// TIA Portal project "FischerTechnik_Origional_program_V16_V17" (V17)

(* hardware
DEVICE "ET 200SP-Station_1"  ET 200SP-Station
   slot 0: "Baugruppenträger_0"  Rack  6ES5 710-8MAx1
   slot 1: "PLC"  CPU 1512SP F-1 PN  6ES7 512-1SK01-0AB0  V2.8
      slot 32768: "PROFINET"  X1
         slot 32771: "Port_3"  X1 P3
   slot 2: "DO1+2"  DQ 16x24VDC/0.5A ST  6ES7 132-6BH01-0BA0  V0.0
      slot 1: "DO1+2"  DQ 16x24VDC/0.5A ST
   slot 3: "DO3+4"  DQ 16x24VDC/0.5A ST  6ES7 132-6BH01-0BA0  V0.0
      slot 1: "DO3+4"  DQ 16x24VDC/0.5A ST
   slot 4: "DO5"  DQ 8x24VDC/0.5A HF  6ES7 132-6BF00-0CA0  V2.0
      slot 1: "DO5"  DQ 8x24VDC/0.5A HF
   slot 5: "DO6"  DQ 8x24VDC/0.5A HF  6ES7 132-6BF00-0CA0  V2.0
      slot 1: "DO6"  DQ 8x24VDC/0.5A HF
   slot 6: "DO7-14"  DQ 4x24VDC/2A HS  6ES7 132-6BD20-0DA0  V2.0
      slot 1: "DO7-14"  DQ 4x24VDC/2A HS
   slot 7: "DO15-22"  DQ 4x24VDC/2A HS  6ES7 132-6BD20-0DA0  V2.0
      slot 1: "DO15-22"  DQ 4x24VDC/2A HS
   slot 8: "DO23-30"  DQ 4x24VDC/2A HS  6ES7 132-6BD20-0DA0  V2.0
      slot 1: "DO23-30"  DQ 4x24VDC/2A HS
   slot 9: "DI1+2"  DI 16x24VDC ST  6ES7 131-6BH01-0BA0  V0.0
      slot 1: "DI1+2"  DI 16x24VDC ST
   slot 10: "DI3"  DI 8x24VDC HF  6ES7 131-6BF00-0CA0  V2.0
      slot 1: "DI3"  DI 8x24VDC HF
   slot 11: "DI4"  DI 8x24VDC HF  6ES7 131-6BF00-0CA0  V2.0
      slot 1: "DI4"  DI 8x24VDC HF
   slot 12: "DI5"  DI 8x24VDC HS  6ES7 131-6BF00-0DA0  V1.0
      slot 1: "DI5"  DI 8x24VDC HS
   slot 13: "DI6"  DI 8x24VDC HS  6ES7 131-6BF00-0DA0  V1.0
      slot 1: "DI6"  DI 8x24VDC HS
   slot 14: "AI7-10"  AI 2xU ST  6ES7 134-6FB00-0BA1  V1.0
      slot 1: "AI7-10"  AI 2xU ST
   slot 15: "End"  Server module  6ES7 193-6PA00-0AA0  V1.1
      slot 1: "End"  Server module
   slot 127: "BA 2xRJ45"  BA 2xRJ45  6ES7 193-6AR00-0AA0  V0.0
      slot 32769: "Port_1"  X1 P1  6ES7 193-6AR00-0AA0
      slot 32770: "Port_2"  X1 P2  6ES7 193-6AR00-0AA0
*)

// ===== PLC "PLC"  CPU 1512SP F-1 PN =====

VAR_GLOBAL   // PLC tag table "HBW - Automated High-Bay Warehouse"
   "IX_HBW_RefSwitchHorizontalAxis_I1" AT %I1.0 : Bool;   // HBW - I1 = Reference switch horizontal axis
   "IX_HBW_LightBarrierInside_I2" AT %I1.1 : Bool;   // HBW - I2 = Light barrier inside
   "IX_HBW_LightBarrierOutside_I3" AT %I1.2 : Bool;   // HBW - I3 = Light barrier outside
   "IX_HBW_RefSwitchVerticalAxis_I4" AT %I1.3 : Bool;   // HBW - I4 = Reference switch vertical axis
   "IX_HBW_TrailSensor1Lower_A1" AT %I5.0 : Bool;   // HBW - A1 = Trail sensor (signal 1, lower)
   "IX_HBW_TrailSensor2Upper_A2" AT %I5.4 : Bool;   // HBW - A2 = Trail sensor (signal 2, upper)
   "IX_HBW_EncoderVerticalAxisImp1_B3" AT %I5.2 : Bool;   // HBW - B3 = Encoder vertical axis imulse 1
   "IX_HBW_EncoderVerticalAxisImp2_B4" AT %I5.6 : Bool;   // HBW - B4 = Encoder vertical axis imulse 2
   "IX_HBW_EncoderHorizontalAxisImp1_B1" AT %I5.1 : Bool;   // HBW - B1 = Encoder horizontal axis imulse 1
   "IX_HBW_EncoderHorizontalAxisImp2_B2" AT %I5.5 : Bool;   // HBW - B2 = Encoder horizontal axis imulse 2
   "IX_HBW_SwitchCantileverFront_I5" AT %I1.4 : Bool;   // HBW - I5 = Reference switch cantilever front
   "IX_HBW_SwitchCantileverBack_I6" AT %I1.5 : Bool;   // HBW - I6 = Reference switch cantilever back
   "QX_HBW_M1_ConveyorBeltForward_Q1" AT %Q1.0 : Bool;   // HBW - Q1 = Motor M1 conveyor belt forward
   "QX_HBW_M1_ConveyorBeltBackward_Q2" AT %Q1.1 : Bool;   // HBW - Q2 = Motor M1 conveyor belt backward
   "QX_HBW_M2_HorizontalTowardsRack_Q3" AT %Q1.2 : Bool;   // HBW - Q3 = Motor M2 horizontal towards rack
   "QX_HBW_M2_HorizontalTowardsConveyorBelt_Q4" AT %Q1.3 : Bool;   // HBW - Q4 = Motor M2 horizontal towards conveyor belt
   "QX_HBW_M3_VerticalAxisDownward_Q5" AT %Q1.4 : Bool;   // HBW - Q5 = Motor M3 vertical axis downward
   "QX_HBW_M3_VerticalAxisUpward_Q6" AT %Q1.5 : Bool;   // HBW - Q6 = Motor M3 vertical axis upward
   "QX_HBW_M4_CantileverForward_Q7" AT %Q1.6 : Bool;   // HBW - Q7 = Motor M4 cantilever forward
   "QX_HBW_M4_CantileverBackward_Q8" AT %Q1.7 : Bool;   // HBW - Q8 = Motor M4 cantilever backward
   "QW_HBW_PWM_ConveyorBelt_M1" AT %QW7 : Int;   // HBW = PWM Motor M1 conveyor belt
   "QW_HBW_PWM_HorizontalAxis_M2" AT %QW9 : Int;   // HBW = PWM Motor M2 horizontal axis
   "QW_HBW_PWM_VerticalAxis_M3" AT %QW11 : Int;   // HBW = PWM Motor M3 vertical axis
   "QW_HBW_PWM_Cantilever_M4" AT %QW13 : Int;   // HBW = PWM Motor M4 cantilever
END_VAR

VAR_GLOBAL   // PLC tag table "MPO - Multi Processing Station with Oven"
   "IX_MPO_RefSwitchTurnTable_PosVac_I1" AT %I1.7 : Bool;   // MPO - I1 = Reference switch turn-table (position vacuum)
   "IX_MPO_RefSwitchTurnTable_PosBelt_I2" AT %I2.0 : Bool;   // MPO - I2 = Reference switch turn-table (position belt)
   "IX_MPO_LightBarrierEndOfConBelt_I3" AT %I2.1 : Bool;   // MPO - I3 = Light barrier end of conveyor belt
   "IX_MPO_RefSwitchTurnTable_PosSaw_I4" AT %I2.2 : Bool;   // MPO - I4 = Reference switch turn-table (position saw)
   "IX_MPO_RefSwitchVac_PosTurnTable_I5" AT %I2.3 : Bool;   // MPO - I5 = Reference switch vacuum (position turn-table)
   "IX_MPO_RefSwitchOvenFeederInside_I6" AT %I2.4 : Bool;   // MPO - I6 = Reference switch oven feeder inside
   "IX_MPO_RefSwitchOvenFeederOutside_I7" AT %I2.5 : Bool;   // MPO - I7 = Reference switch oven feeder outside
   "IX_MPO_RefSwitchVac_PosOven_I8" AT %I2.6 : Bool;   // MPO - I8 = Reference switch vacuum (position oven)
   "IX_MPO_LightBarrierOven_I9" AT %I2.7 : Bool;   // MPO - I9 = Light barrier oven
   "QX_MPO_M1_TurnTableClockwise_Q1" AT %Q3.0 : Bool;   // MPO - Q1 = Motor M1 turn-table clockwise
   "QX_MPO_M1_TurnTableCounterclockwise_Q2" AT %Q3.1 : Bool;   // MPO - Q2 = Motor M1 turn-table counterclockwise
   "QX_MPO_M2_ConveyorBeltForward_Q3" AT %Q3.2 : Bool;   // MPO - Q3 = Motor M2 conveyor belt forward
   "QX_MPO_M3_Saw_Q4" AT %Q3.3 : Bool;   // MPO - Q4 = Motor M3 saw
   "QX_MPO_M4_OvenFeederRetract_Q5" AT %Q3.4 : Bool;   // MPO - Q5 = Motor M4 oven feeder retract
   "QX_MPO_M4_OvenFeederExtend_Q6" AT %Q3.5 : Bool;   // MPO - Q6 = Motor M4 oven feeder extend
   "QX_MPO_M5_VacuumTowardsOven_Q7" AT %Q3.6 : Bool;   // MPO - Q7 = Motor M5 vacuum towards oven
   "QX_MPO_M5_VacuumTowardsTurnTable_Q8" AT %Q3.7 : Bool;   // MPO - Q8 = Motor M5 vacuum towards turn-table
   "QX_MPO_LightOven_Q9" AT %Q4.0 : Bool;   // MPO - Q9 = Light oven
   "QX_MPO_Compressor_Q10" AT %Q4.1 : Bool;   // MPO - Q10 = Compressor
   "QX_MPO_ValveVacuum_Q11" AT %Q4.2 : Bool;   // MPO - Q11 = Valve vacuum
   "QX_MPO_ValveLowering_Q12" AT %Q4.3 : Bool;   // MPO - Q12 = Valve lowering
   "QX_MPO_ValveOvenDoor_Q13" AT %Q4.4 : Bool;   // MPO - Q13 = Valve oven door
   "QX_MPO_ValveFeeder_Q14" AT %Q4.5 : Bool;   // MPO - Q14 = Valve feeder
   "QW_MPO_PWM_TurnTable_M1" AT %QW23 : Int;   // MPO = PWM Motor M1 turn-table
   "QW_MPO_PWM_Vacuum_M5" AT %QW25 : Int;   // MPO = PWM Motor M5 turn-table
END_VAR

VAR_GLOBAL   // PLC tag table "VGR - Vacuum Gripper Robot"
   "IX_VGR_RefSwitchVerticalAxis_I1" AT %I1.6 : Bool;   // VGR - I1 = Reference switch vertical axis
   "IX_VGR_RefSwitchHorizontalAxis_I2" AT %I3.6 : Bool;   // VGR - I2 = Reference switch horizontal axis
   "IX_VGR_RefSwitchRotate_I3" AT %I3.7 : Bool;   // VGR - I3 = Reference switch rotate
   "IX_VGR_EncoderVerticalAxisImp1_B1" AT %I6.0 : Bool;   // VGR - B1 = Encoder vertical axis imulse 1
   "IX_VGR_EncoderVerticalAxisImp2_B2" AT %I6.4 : Bool;   // VGR - B2 = Encoder vertical axis imulse 2
   "IX_VGR_EncoderHorizontalAxisImp1_B3" AT %I6.1 : Bool;   // VGR - B3 = Encoder horizontal axis imulse 1
   "IX_VGR_EncoderHorizontalAxisImp2_B4" AT %I6.5 : Bool;   // VGR - B4 = Encoder horizontal axis imulse 2
   "IX_VGR_EncoderRotateImp1_B5" AT %I6.2 : Bool;   // VGR - B5 = Encoder rotate impulse 1
   "IX_VGR_EncoderRotateImp2_B6" AT %I6.6 : Bool;   // VGR - B6 = Encoder rotate impulse 2
   "QX_VGR_M1_VerticalAxisUp_Q1" AT %Q2.0 : Bool;   // VGR - Q1 = Motor M1 vertical axis up
   "QX_VGR_M1_VerticalAxisDown_Q2" AT %Q2.1 : Bool;   // VGR - Q2 = Motor M1 vertical axis down
   "QX_VGR_M2_HorizontalAxisBackward_Q3" AT %Q2.2 : Bool;   // VGR - Q3 = Motor M2 horizontal axis backward
   "QX_VGR_M2_HorizontalAxisForward_Q4" AT %Q2.3 : Bool;   // VGR - Q4 = Motor M2 horizontal axis forward
   "QX_VGR_M3_RotateClockwise_Q5" AT %Q2.4 : Bool;   // VGR - Q5 = Motor M3 rotate clockwise
   "QX_VGR_M3_RotateCounterclockwise_Q6" AT %Q2.5 : Bool;   // VGR - Q6 = Motor M3 rotate counterclockwise
   "QX_VGR_Compressor_Q7" AT %Q2.6 : Bool;   // VGR - Q7 = Compressor
   "QX_VGR_ValveVacuum_Q8" AT %Q2.7 : Bool;   // VGR - Q8 = Valve vacuum
   "QW_VGR_PWM_Vertical_M1" AT %QW15 : Int;   // VGR = PWM Motor M1 vertical axis
   "QW_VGR_PWM_Horizontal_M2" AT %QW17 : Int;   // VGR = PWM Motor M2 horizontal axis
   "QW_VGR_PWM_Rotate_M3" AT %QW19 : Int;   // VGR = PWM Motor M3 rotate axis
END_VAR

VAR_GLOBAL   // PLC tag table "SLD - Sorting Line with Detection"
   "IX_SLD_PulseCounter_I1" AT %I3.0 : Bool;   // SLD - I1 = Pulse counter
   "IX_SLD_LightBarrierInlet_I2" AT %I3.1 : Bool;   // SLD - I2 = Light barrier inlet
   "IX_SLD_LightBarrierBehindColorSensor_I3" AT %I3.2 : Bool;   // SLD - I3 = Light barrier behind color sensor
   "IW_SLD_ColorSensor_A4" AT %IW7 : Word;   // SLD - A4 = Color sensor
   "IX_SLD_LightBarrierWhite_I5" AT %I3.3 : Bool;   // SLD - I5 = Light barrier white
   "IX_SLD_LightBarrierRed_I6" AT %I3.4 : Bool;   // SLD - I6 = Light barrier red
   "IX_SLD_LightBarrierBlue_I7" AT %I3.5 : Bool;   // SLD - I7 = Light barrier blue
   "QX_SLD_M1_ConveyorBelt_Q1" AT %Q5.0 : Bool;   // SLD - Q1 = Motor M1conveyor belt
   "QX_SLD_Compressor_Q2" AT %Q5.1 : Bool;   // SLD - Q2 = Compressor
   "QX_SLD_ValveFirstEjectorWhite_Q3" AT %Q5.2 : Bool;   // SLD - Q3 = Valve first ejector (white)
   "QX_SLD_ValveSecondEjectorRed_Q4" AT %Q5.3 : Bool;   // SLD - Q4 = Valve second ejector (red)
   "QX_SLD_ValveThirdEjectorBlue_Q5" AT %Q5.4 : Bool;   // SLD - Q5 = Valve third ejector (blue)
END_VAR

VAR_GLOBAL   // PLC tag table "SSC - Sensor-Station Camera"
   "IX_SSC_RefSwitchVerticalAxis_I1" AT %I4.0 : Bool;   // SSC - I1 = Reference switch vertical axis
   "IX_SSC_RefSwitchHorizontalAxis_I2" AT %I4.1 : Bool;   // SSC - I2 = Reference switch horizontal axis
   "IX_SSC_LightBarrierStorage_I3" AT %I4.3 : Bool;   // SSC - I3 = Light barrier inlet
   "IX_SSC_LightBarrierOutsourcing_I4" AT %I4.2 : Bool;   // SSC - I4 = Light barrier behind color sensor
   "IW_SSC_ColorSensor_A1" AT %IW9 : Word;   // SSC - A1 = Color sensor
   "IX_SSC_EncoderVerticalAxisImp1_B1" AT %I5.3 : Bool;   // SSC - B1 = Encoder vertical axis imulse 1
   "IX_SSC_EncoderVerticalAxisImp2_B2" AT %I5.7 : Bool;   // SSC - B2 = Encoder vertical axis imulse 2
   "IX_SSC_EncoderHorizontalAxisImp1_B3" AT %I6.3 : Bool;   // SSC - B3 = Encoder horizontal axis imulse 1
   "IX_SSC_EncoderHorizontalAxisImp2_B4" AT %I6.7 : Bool;   // SSC - B4 = Encoder horizontal axis imulse 2
   "QX_SSC_M1_VerticalAxisUp_Q1" AT %Q6.0 : Bool;   // SSC - Q1 = Motor M1 vertical axis up
   "QX_SSC_M1_VerticalAxisDown_Q2" AT %Q6.1 : Bool;   // SSC - Q2 = Motor M1 vertical axis down
   "QX_SSC_M2_HorizontalAxisClockwise_Q3" AT %Q6.3 : Bool;   // SSC - Q3 = Motor M2 horizontal axis backward
   "QX_SSC_M2_HorizontalAxisCounterclockwise_Q4" AT %Q6.2 : Bool;   // SSC - Q4 = Motor M2 horizontal axis forward
   "QX_SSC_LED_Green_Q5" AT %Q6.4 : Bool;   // SSC - Q5 = LED Green
   "QX_SSC_LED_Yellow_Q6" AT %Q6.5 : Bool;   // SSC - Q6 = LED Yellow
   "QX_SSC_LED_Red_Q7" AT %Q6.6 : Bool;   // SSC - Q7 = LED Red
   "QX_SSC_LED_Red_Online_Q8" AT %Q6.7 : Bool;   // SSC - Q8 = LED Red Online
   "QW_SSC_PWM_Vertical_M1" AT %QW27 : Int;   // SSC = PWM Motor M1 vertical axis
   "QW_SSC_PWM_Horizontal_M2" AT %QW29 : Int;   // SSC = PWM Motor M2 horizontal axis
END_VAR

VAR_GLOBAL   // PLC tag table "Global"
   "IX_Set_Park_Position" AT %I4.7 : Bool;
END_VAR

VAR_GLOBAL   // PLC tag table "Variablentabelle aus XML_1"
   "IX_Fill_HBW" AT %I4.6 : Bool;
END_VAR

TYPE "typ_MQTT_Interface_Dashboard"
VERSION : 0.1
   STRUCT
      Subscribe : "typ_MQTT_Interface_Dashboard_Subscribe";
      Publish : "typ_MQTT_ Interface_Dashboard_Publish";
   END_STRUCT;
END_TYPE

TYPE "typ_Stock_Item"
VERSION : 0.1
   STRUCT
      ldt_ts : LDT;
      StockItem : Array[1..3, 1..3] of "typ_Workpiece";
      s_location : String;
   END_STRUCT;
END_TYPE

TYPE "typ_Acknowledgment_Client"
VERSION : 0.1
   STRUCT
      ldt_ts : LDT;
      i_code : Int;
      Workpiece : "typ_Workpiece";
   END_STRUCT;
END_TYPE

TYPE "typ_State_Client"
VERSION : 0.1
   STRUCT
      ldt_ts : LDT;
      s_station : String;
      i_code : Int;
      s_description : String;
      x_active : Bool;
      s_target : String;
   END_STRUCT;
END_TYPE

TYPE "typ_Broadcast"
VERSION : 0.1
   STRUCT
      ldt_ts : LDT;
      di_hardwareId : DInt;
      di_hardwareModel : DInt;
      s_softwareName : String;
      di_softwareVersion : DInt;
      s_message : String;
   END_STRUCT;
END_TYPE

TYPE "typ_Config_Camera_Picture"
VERSION : 0.1
   STRUCT
      ldt_ts : LDT;
      di_period : DInt;
   END_STRUCT;
END_TYPE

TYPE "typ_Config_Brightness_Sensor"
VERSION : 0.1
   STRUCT
      ldt_ts : LDT;
      x_on : Bool;
      i_fps : Int;
   END_STRUCT;
END_TYPE

TYPE "typ_Config_Enviorment_Sensor"
VERSION : 0.1
   STRUCT
      ldt_ts : LDT;
      di_period : DInt;
   END_STRUCT;
END_TYPE

TYPE "typ_History"
VERSION : 0.1
   STRUCT
      ldt_ts : LDT;
      i_code : Int;
   END_STRUCT;
END_TYPE

TYPE "typ_Pos_Pan_Tilt_Unit_Mov"
VERSION : 0.1
   STRUCT
      ldt_ts : LDT;
      s_cmd : String;
      i_degree : Int;
   END_STRUCT;
END_TYPE

TYPE "typ_Workpiece"
VERSION : 0.1
   STRUCT
      s_id : String;
      s_type : String;
      s_state : String;
   END_STRUCT;
END_TYPE

TYPE "typ_Order_Workpiece_Buttons_State"
VERSION : 0.1
   STRUCT
      ldt_ts : LDT;
      s_state : String;
      s_type : String;
   END_STRUCT;
END_TYPE

TYPE "typ_NFC_Module_State"
VERSION : 0.1
   STRUCT
      ldt_ts : LDT;
      Workpiece : "typ_Workpiece";
      History : Array[1..20] of "typ_History";
   END_STRUCT;
END_TYPE

TYPE "typ_VGR"
VERSION : 0.1
   STRUCT
      x_Start_Park_Position : Bool;
      x_Park_Position_Reached : Bool;
      x_NFC_Start_First : Bool;
      x_NFC_Start : Bool;
      x_NFC_Completed : Bool;
      x_HBW_Storage : Bool;
      x_HBW_Outsource : Bool;
      s_HBW_Outsource_Typ : String;
      x_HBW_Discards : Bool;
      x_HBW_PickedUp : Bool;
      x_MPO_Req_Discard : Bool;
      x_MPO_Discards : Bool;
      x_Ready_For_Outsource : Bool;
      x_State_Process : Bool;
      x_Workpiece_NiO : Bool;
      horizontal_Axis : "typ_Axis";
      vertical_Axis : "typ_Axis";
      rotate_Axis : "typ_Axis";
      Workpiece : "typ_Workpiece";
      History : Array[1..20] of "typ_History";
      di_Pos_DSI_horizontal : DInt;
      di_Pos_DSI_Collect_vertical : DInt;
      di_Pos_DSI_Discard_vertical : DInt;
      di_Offset_Pos_DSI_NFC_vertical : DInt;
      di_Pos_DSI_rotate : DInt;
      di_Pos_DSO_horizontal : DInt;
      di_Pos_DSO_Collect_vertical : DInt;
      di_Pos_DSO_Discard_vertical : DInt;
      di_Offset_Pos_DSO_vertical : DInt;
      di_Pos_DSO_rotate : DInt;
      di_Pos_Color_horizontal : DInt;
      di_Pos_Color_vertical : DInt;
      di_Pos_Color_rotate : DInt;
      di_Pos_NFC_horizontal : DInt;
      di_Pos_NFC_vertical : DInt;
      di_Pos_NFC_rotate : DInt;
      di_Pos_MPO_horizontal : DInt;
      di_Pos_MPO_vertical : DInt;
      di_Offset_Pos_MPO_vertical : DInt;
      di_Pos_MPO_rotate : DInt;
      di_Pos_HBW_horizontal : DInt;
      di_Offset_Pos_HBW_horizontal : DInt;
      di_Pos_HBW_Collect_vertical : DInt;
      di_Pos_HBW_Discard_vertical : DInt;
      di_Offset_Pos_HBW_vertical : DInt;
      di_Pos_HBW_rotate : DInt;
      di_Pos_NiO_horizontal : DInt;
      di_Pos_NiO_vertical : DInt;
      di_Pos_NiO_rotate : DInt;
      di_Pos_SLD_Blue_horizontal : DInt;
      di_Pos_SLD_Blue_vertical : DInt;
      di_Pos_SLD_Blue_rotate : DInt;
      di_Pos_SLD_Red_horizontal : DInt;
      di_Pos_SLD_Red_vertical : DInt;
      di_Pos_SLD_Red_rotate : DInt;
      di_Pos_SLD_White_horizontal : DInt;
      di_Pos_SLD_White_vertical : DInt;
      di_Pos_SLD_White_rotate : DInt;
      di_Pos_Park_horizontal : DInt;
      di_Pos_Park_vertical : DInt;
      di_Pos_Park_rotate : DInt;
   END_STRUCT;
END_TYPE

TYPE "typ_SetupAxis"
VERSION : 0.1
   STRUCT
      x_Setup_Activ : Bool;   // Set up calibration active
      i_AxisSelection : Int;   // Number of the axis
      i_Function : Int;   // 0 = automatic, 10 = ref. Travel, 20 = tap, 30 = tap with step width, 40 = start
      x_Set_Ref_Pos : Bool;   // Set reference value
      x_Set_Soft_End_Pos : Bool;   // Set software end positions
      x_Approach_Ref_Pos : Bool;   // Approach reference
      x_Axis_Pos : Bool;   // Axis positiv
      x_Axis_Neg : Bool;   // Axis negative
      x_Approach_Target_Pos : Bool;   // Approach Target position
      w_Increment : Word;   // Increments per step
      i_PWM : Int;   // PWM Signal
      di_Target_Position : DInt;   // Target position
      di_ActualPosition : DInt;   // Actual position
      di_Ref_Pos : DInt;   // Reference position
      di_Actual_Ref_Pos : DInt;   // Current reference position
      di_Soft_End_Pos_Neg : DInt;   // Software end position negative
      di_Actual_Soft_End_Pos_Neg : DInt;   // Current software end position negative
      di_Soft_End_Pos_Pos : DInt;   // Software end position positiv
      di_Actual_Soft_End_Pos_Pos : DInt;   // Current software end position positiv
      di_LoopValue : DInt;   // Loop value
   END_STRUCT;
END_TYPE

TYPE "typ_Axis_Data"
VERSION : 0.1
   STRUCT
      di_Pos_Soft_Switch : DInt := 0;
      di_Neg_Soft_Switch : DInt := 0;
      di_Ref_Pos : DInt := 0;
      di_Loop_Value : DInt := 0;
      di_Pos_Window : DInt := 15;
   END_STRUCT;
END_TYPE

TYPE "typ_Axis"
VERSION : 0.1
   STRUCT
      x_Start_Positioning : Bool;
      x_Reference : Bool;
      x_Referenced : Bool;
      x_Position_Reached : Bool;
      di_Target_Position : DInt;
      di_Increment : DInt;
      di_Actual_Position : DInt := 0;
      i_PWM : Int;
      Config : "typ_Axis_Data";
   END_STRUCT;
END_TYPE

TYPE "typ_SSC"
VERSION : 0.1
   STRUCT
      x_Start_Park_Position : Bool;
      x_Park_Position_Reached : Bool;
      x_Error : Bool;
      di_Pos_Centre_Horizontal : DInt;
      di_Pos_Centre_Vertical : DInt;
      di_Pos_HBW_Horizontal : DInt;
      di_Pos_HBW_Vertical : DInt;
      di_Pos_Park_Horizontal : DInt;
      di_Pos_Park_Vertical : DInt;
      w_Threshold_White_Red : Word;
      w_Threshold_Red_Blue : Word;
      Horizontal_Axis : "typ_Axis";
      Vertical_Axis : "typ_Axis";
      Workpiece : "typ_Workpiece";
      History : Array[1..20] of "typ_History";
   END_STRUCT;
END_TYPE

TYPE "typ_HBW"
VERSION : 0.1
   STRUCT
      x_Start_Park_Position : Bool;
      x_Park_Position_Reached : Bool;
      x_HBW_PickedUp_Accepted : Bool;
      x_HBW_Discards_Accepted : Bool;
      x_HBW_PickUp_Ready : Bool;
      x_HBW_Container_Available : Bool;
      x_Error : Bool;
      di_PosBelt_Horizontal : DInt;
      di_PosBelt_Vertical : DInt;
      di_Offset_Pos_Belt_Vertical : DInt;
      di_PosRack_A1_Horizontal : DInt;
      di_PosRack_A1_Vertical : DInt;
      di_PosRack_B2_Horizontal : DInt;
      di_PosRack_B2_Vertical : DInt;
      di_PosRack_C3_Horizontal : DInt;
      di_PosRack_C3_Vertical : DInt;
      di_Offset_Pos_Rack_Vertical : DInt;
      di_Pos_Park_Horizontal : DInt;
      di_Pos_Park_Vertical : DInt;
      i_PWM_ConveyorBelt : Int := 800;
      i_PWM_Cantilever : Int := 800;
      Workpiece : "typ_Workpiece";
      History : Array[1..20] of "typ_History";
      Rack_Pos : Array[1..3, 1..3] of "typ_Rack_Pos";
      Rack_Workpiece : Array[1..3, 1..3] of "typ_Workpiece";
      Rack_History : Array[1..3, 1..3] of "typ_Rack_History";
      Horizontal_Axis : "typ_Axis";
      Vertical_Axis : "typ_Axis";
   END_STRUCT;
END_TYPE

TYPE "typ_MQTT_ Interface_Dashboard_Publish"
VERSION : 0.1
   STRUCT
      ldt_AcknowledgeButton : LDT;
      ConfigRateEnviormentSensor : "typ_Config_Enviorment_Sensor";
      ConfigRateBrightnessSensor : "typ_Config_Brightness_Sensor";
      ConfigRateCameraPicture : "typ_Config_Camera_Picture";
      PosPanTiltUnit : "typ_Pos_Pan_Tilt_Unit_Mov";
      OrderWorkpieceButton : "typ_Order_Workpiece_Buttons";
      ActionButtonNFCModule : "typ_Action_Buttons_NFC_Module";
   END_STRUCT;
END_TYPE

TYPE "typ_MQTT_Interface_Dashboard_Subscribe"
VERSION : 0.1
   STRUCT
      EnvironmentSensor : "typ_Environment_Sensor";
      BrightnessSensor : "typ_Brightness_Sensor";
      CameraPicture : "typ_Camera_Picture";
      PosPanTiltUnit : "typ_Pos_Pan_Tilt_Unit_Enc";
      AlertMessage : "typ_Alert_Message";
      Broadcast : "typ_Broadcast";
      State_HBW : "typ_State_Client";
      State_VGR : "typ_State_Client";
      State_MPO : "typ_State_Client";
      State_SLD : "typ_State_Client";
      State_DSI : "typ_State_Client";
      State_DSO : "typ_State_Client";
      Stock_HBW : "typ_Stock_Item";
      State_Order : "typ_Order_Workpiece_Buttons_State";
      State_NFC_Device : "typ_NFC_Module_State";
   END_STRUCT;
END_TYPE

TYPE "typ_Rack_Pos"
VERSION : 0.1
   STRUCT
      di_PosRack_Horizontal : DInt;
      di_PosRack_Vertical : DInt;
   END_STRUCT;
END_TYPE

TYPE "typ_VGR_Trigger"
VERSION : 0.1
   STRUCT
      ldt_ts : LDT;
      i_code : Int;
      Workpiece : "typ_Workpiece";
   END_STRUCT;
END_TYPE

TYPE "typ_Alert_Message"
VERSION : 0.1
   STRUCT
      ldt_ts : LDT;
      s_id : String;
      s_data : String;
      i_code : Int;
   END_STRUCT;
END_TYPE

TYPE "typ_Camera_Picture"
VERSION : 0.1
   STRUCT
      ldt_ts : LDT;
      s_data : String;
   END_STRUCT;
END_TYPE

TYPE "typ_Pos_Pan_Tilt_Unit_Enc"
VERSION : 0.1
   STRUCT
      ldt_ts : LDT;
      r_pan : Real;
      r_tilt : Real;
   END_STRUCT;
END_TYPE

TYPE "typ_Brightness_Sensor"
VERSION : 0.1
   STRUCT
      ldt_ts : LDT;
      r_br : Real;
      i_ldr : Int;
   END_STRUCT;
END_TYPE

TYPE "typ_Environment_Sensor"
VERSION : 0.1
   STRUCT
      ldt_ts : LDT;
      r_t : Real;
      r_rt : Real;
      r_h : Real;
      r_rh : Real;
      r_p : Real;
      i_iaq : Int;
      i_aq : Int;
      di_gr : DInt;
   END_STRUCT;
END_TYPE

TYPE "typ_Order_Workpiece_Buttons"
VERSION : 0.1
   STRUCT
      ldt_ts : LDT;
      s_type : String;
   END_STRUCT;
END_TYPE

TYPE "typ_Action_Buttons_NFC_Module"
VERSION : 0.1
   STRUCT
      ldt_ts : LDT;
      s_cmd : String;
   END_STRUCT;
END_TYPE

TYPE "typ_Joysticks"
VERSION : 0.1
   STRUCT
      ldt_ts : LDT;
      r_br : Real;
      i_ldr : Int;
   END_STRUCT;
END_TYPE

TYPE "typ_MPO"
VERSION : 0.1
   STRUCT
      x_Start_Park_Position : Bool;
      x_Park_Position_Reached : Bool;
      x_Discard_Ready : Bool;
      x_MPO_Discards_Accepted : Bool;
      x_Error : Bool;
      i_PWM_TurnTable : Int := 700;
      i_PWM_Vacuum : Int := 1000;
      Workpiece : "typ_Workpiece";
      History : Array[1..20] of "typ_History";
   END_STRUCT;
END_TYPE

TYPE "typ_SLD"
VERSION : 0.1
   STRUCT
      x_Error : Bool;
      i_CounterValue_Blue : Int := 8;
      i_CounterValue_White : Int := 2;
      i_CounterValue_Red : Int := 4;
      i_Counter_Actual : Int;
      w_Threshold_White_Red : Word;
      w_Threshold_Red_Blue : Word;
      Workpiece : "typ_Workpiece";
      History : Array[1..20] of "typ_History";
   END_STRUCT;
END_TYPE

TYPE "typ_Setup"
VERSION : 0.1
   STRUCT
      r_Version_SPS : Real := 1.4;
      x_Fill_Rack_HBW : Bool;
      x_Start_TON_Fill_HBW : Bool;
      x_Clean_Rack_HBW : Bool;
      x_Park_Position : Bool;
      x_AcknowledgeButton : Bool;
      x_Color_Sensor_Calibration : Bool;
      x_Set_Calib_Value_Color_Blue : Bool;
      x_Set_Calib_Value_Color_White : Bool;
      x_Set_Calib_Value_Color_Red : Bool;
      x_Calculate_Value_Color : Bool;
      i_Color_Sensor_Selection : Int;
      w_Calib_ColorValue_Blue : Word;
      w_Calib_ColorValue_White : Word;
      w_Calib_ColorValue_Red : Word;
      w_Threshold_White_Red : Word;
      w_Threshold_Red_Blue : Word;
      w_Actual_ColorValue : Word;
      x_Set_Pos_Activ : Bool;   // Set up calibration active
      x_Start_Positioning : Bool;
      x_Final_Positioning : Bool;
      x_Home_Positioning : Bool;
      x_Start_Offset : Bool;
      i_Pos_Selection : Int;   // Number of the axis
      di_Pos_Horizontal : DInt;
      di_Pos_Vertical : DInt;
      di_Pos_Rotate : DInt;
      x_Counter_Value_Calibration : Bool;
      i_Calib_CounterValue_Blue : Int := 26;
      i_Calib_CounterValue_White : Int := 5;
      i_Calib_CounterValue_Red : Int := 16;
      x_Set_CounterValues : Bool;
      x_Activate_Continuous_Operation : Bool;
   END_STRUCT;
END_TYPE

TYPE "typ_Rack_History"
VERSION : 0.1
   STRUCT
      History : Array[1..20] of "typ_History";
   END_STRUCT;
END_TYPE

TYPE "typ_MQTT_Interface_TXT_Controller"
VERSION : 0.1
   STRUCT
      Subscribe : "typ_MQTT_Interface_TXT_Controler_Subscribe";
      Publish : "typ_MQTT_ Interface_TXT_Controler_Publish";
   END_STRUCT;
END_TYPE

TYPE "typ_SPS_NFC_Module_State"
VERSION : 0.1
   STRUCT
      ldt_ts : LDT;
      Workpiece : "typ_Workpiece";
      History : Array[1..20] of "typ_History";
   END_STRUCT;
END_TYPE

TYPE "typ_MQTT_ Interface_TXT_Controler_Publish"
VERSION : 0.1
   STRUCT
      ActionButtonNFCModule : "typ_SPS_Action_Buttons_NFC_Module";
   END_STRUCT;
END_TYPE

TYPE "typ_MQTT_Interface_TXT_Controler_Subscribe"
VERSION : 0.1
   STRUCT
      State_NFC_Device : "typ_SPS_NFC_Module_State";
   END_STRUCT;
END_TYPE

TYPE "typ_SPS_Action_Buttons_NFC_Module"
VERSION : 0.1
   STRUCT
      ldt_ts : LDT;
      s_cmd : String;
      Workpiece : "typ_Workpiece";
      History : Array[1..20] of "typ_History";
   END_STRUCT;
END_TYPE

DATA_BLOCK "gtyp_Interface_Dashboard"   // DB1
TITLE = Global Interface Dashboard Cloud
{ S7_Optimized_Access := 'TRUE' }
AUTHOR : A.Schaefer
VERSION : 0.0
BEGIN
END_DATA_BLOCK

DATA_BLOCK "gtyp_VGR"   // DB2
TITLE = Global DB VGR
{ S7_Optimized_Access := 'TRUE' }
AUTHOR : A.Schaefer
VERSION : 0.0
BEGIN
   horizontal_Axis.i_PWM := 500;
   horizontal_Axis.Config.di_Pos_Soft_Switch := 20000;
   vertical_Axis.i_PWM := 800;
   vertical_Axis.Config.di_Pos_Soft_Switch := 20000;
   rotate_Axis.i_PWM := 500;
   rotate_Axis.Config.di_Pos_Soft_Switch := 20000;
   di_Pos_DSI_horizontal := 20;
   di_Pos_DSI_Collect_vertical := 2950;
   di_Offset_Pos_DSI_NFC_vertical := 1200;
   di_Pos_DSI_rotate := 30;
   di_Pos_DSO_horizontal := 2070;
   di_Pos_DSO_Discard_vertical := 1480;
   di_Offset_Pos_DSO_vertical := 500;
   di_Pos_DSO_rotate := 970;
   di_Pos_Color_horizontal := 150;
   di_Pos_Color_vertical := 2450;
   di_Pos_Color_rotate := 430;
   di_Pos_NFC_horizontal := 900;
   di_Pos_NFC_vertical := 2450;
   di_Pos_NFC_rotate := 700;
   di_Pos_MPO_horizontal := 3400;
   di_Pos_MPO_vertical := 1800;
   di_Offset_Pos_MPO_vertical := 650;
   di_Pos_MPO_rotate := 3500;
   di_Pos_HBW_horizontal := 600;
   di_Pos_HBW_Collect_vertical := 650;
   di_Pos_HBW_Discard_vertical := 200;
   di_Offset_Pos_HBW_vertical := 100;
   di_Pos_HBW_rotate := 5350;
   di_Pos_NiO_vertical := 2700;
   di_Pos_NiO_rotate := 1100;
   di_Pos_SLD_Blue_horizontal := 2150;
   di_Pos_SLD_Blue_vertical := 3100;
   di_Pos_SLD_Blue_rotate := 1200;
   di_Pos_SLD_Red_horizontal := 1580;
   di_Pos_SLD_Red_vertical := 3100;
   di_Pos_SLD_Red_rotate := 1460;
   di_Pos_SLD_White_horizontal := 1370;
   di_Pos_SLD_White_vertical := 3100;
   di_Pos_SLD_White_rotate := 1770;
   di_Pos_Park_horizontal := 150;
   di_Pos_Park_vertical := 3000;
   di_Pos_Park_rotate := 1750;
END_DATA_BLOCK

DATA_BLOCK "PRG_SSC_Axis_Vertical_DB"   // DB3
{ S7_Optimized_Access := 'TRUE' }
AUTHOR : A.Schaefer
VERSION : 0.1
// stored: InstanceOfName PRG_SSC_Axis_Vertical
"PRG_SSC_Axis_Vertical"
BEGIN
END_DATA_BLOCK

DATA_BLOCK "gtyp_SetupAxis"   // DB4
TITLE = Global DB Setup Axis
{ S7_Optimized_Access := 'TRUE' }
AUTHOR : A.Schaefer
VERSION : 0.0
BEGIN
END_DATA_BLOCK

DATA_BLOCK "PRG_MPO_Ablauf_DB"   // DB5
{ S7_Optimized_Access := 'TRUE' }
AUTHOR : A.Schaefer
VERSION : 0.1
// stored: InstanceOfName PRG_MPO_Ablauf
"PRG_MPO_Ablauf"
BEGIN
END_DATA_BLOCK

DATA_BLOCK "PRG_SSC_Axis_Vertical_Act_Pos_DB"   // DB6
{ S7_Optimized_Access := 'TRUE' }
AUTHOR : A.Schaefer
VERSION : 0.1
// stored: InstanceOfName PRG_SSC_Axis_Vertical_Act_Pos
"PRG_SSC_Axis_Vertical_Act_Pos"
BEGIN
END_DATA_BLOCK

DATA_BLOCK "PRG_SSC_Axis_Horizontal_DB"   // DB7
{ S7_Optimized_Access := 'TRUE' }
AUTHOR : A.Schaefer
VERSION : 0.1
// stored: InstanceOfName PRG_SSC_Axis_Horizontal
"PRG_SSC_Axis_Horizontal"
BEGIN
END_DATA_BLOCK

DATA_BLOCK "PRG_VGR_Axis_horizontal_DB"   // DB8
{ S7_Optimized_Access := 'TRUE' }
AUTHOR : A.Schaefer
VERSION : 0.1
// stored: InstanceOfName PRG_VGR_Axis_horizontal
"PRG_VGR_Axis_horizontal"
BEGIN
END_DATA_BLOCK

DATA_BLOCK "PRG_VGR_Axis_vertical_DB"   // DB9
{ S7_Optimized_Access := 'TRUE' }
AUTHOR : A.Schaefer
VERSION : 0.1
// stored: InstanceOfName PRG_VGR_Axis_vertical
"PRG_VGR_Axis_vertical"
BEGIN
END_DATA_BLOCK

DATA_BLOCK "PRG_VGR_Axis_rotate_DB"   // DB10
{ S7_Optimized_Access := 'TRUE' }
AUTHOR : A.Schaefer
VERSION : 0.1
// stored: InstanceOfName PRG_VGR_Axis_rotate
"PRG_VGR_Axis_rotate"
BEGIN
END_DATA_BLOCK

DATA_BLOCK "gtyp_MPO"   // DB11
TITLE = Global DB MPO
{ S7_Optimized_Access := 'TRUE' }
AUTHOR : A.Schaefer
VERSION : 0.0
BEGIN
   i_PWM_TurnTable := 1000;
END_DATA_BLOCK

DATA_BLOCK "PRG_NFC_DB"   // DB12
{ S7_Optimized_Access := 'TRUE' }
AUTHOR : A.Schaefer
VERSION : 0.1
// stored: InstanceOfName PRG_NFC
"PRG_NFC"
BEGIN
END_DATA_BLOCK

DATA_BLOCK "gtyp_SSC"   // DB13
TITLE = Global DB SSC
{ S7_Optimized_Access := 'TRUE' }
AUTHOR : A.Schaefer
VERSION : 0.0
BEGIN
   di_Pos_Centre_Horizontal := 3000;
   di_Pos_Centre_Vertical := 1400;
   di_Pos_HBW_Horizontal := 5400;
   di_Pos_HBW_Vertical := 950;
   di_Pos_Park_Horizontal := 3000;
   di_Pos_Park_Vertical := 200;
   w_Threshold_White_Red := 16#25DA;
   w_Threshold_Red_Blue := 16#4F32;
   Horizontal_Axis.i_PWM := 1000;
   Horizontal_Axis.Config.di_Pos_Soft_Switch := 5450;
   Horizontal_Axis.Config.di_Pos_Window := 25;
   Vertical_Axis.i_PWM := 1000;
   Vertical_Axis.Config.di_Pos_Soft_Switch := 3000;
   Vertical_Axis.Config.di_Pos_Window := 25;
END_DATA_BLOCK

DATA_BLOCK "PRG_HBW_Axis_Vertical_DB"   // DB14
{ S7_Optimized_Access := 'TRUE' }
AUTHOR : A.Schaefer
VERSION : 0.1
// stored: InstanceOfName PRG_HBW_Axis_Vertical
"PRG_HBW_Axis_Vertical"
BEGIN
END_DATA_BLOCK

DATA_BLOCK "PRG_VGR_Axis_horizontal_Act_Pos_DB"   // DB15
{ S7_Optimized_Access := 'TRUE' }
AUTHOR : A.Schaefer
VERSION : 0.1
// stored: InstanceOfName PRG_VGR_Axis_horizontal_Act_Pos
"PRG_VGR_Axis_horizontal_Act_Pos"
BEGIN
END_DATA_BLOCK

DATA_BLOCK "PRG_SSC_Ablauf_DB"   // DB16
{ S7_Optimized_Access := 'TRUE' }
AUTHOR : A.Schaefer
VERSION : 0.1
// stored: InstanceOfName PRG_SSC_Ablauf
"PRG_SSC_Ablauf"
BEGIN
END_DATA_BLOCK

DATA_BLOCK "gtyp_HBW"   // DB17
TITLE = Global DB HBW
{ S7_Optimized_Access := 'TRUE' }
AUTHOR : A.Schaefer
VERSION : 0.0
BEGIN
   di_PosBelt_Horizontal := 18;
   di_PosBelt_Vertical := 2800;
   di_Offset_Pos_Belt_Vertical := 370;
   di_PosRack_A1_Horizontal := 2870;
   di_PosRack_A1_Vertical := 400;
   di_PosRack_B2_Horizontal := 5200;
   di_PosRack_B2_Vertical := 1750;
   di_PosRack_C3_Horizontal := 7560;
   di_PosRack_C3_Vertical := 3250;
   di_Offset_Pos_Rack_Vertical := 370;
   di_Pos_Park_Horizontal := 600;
   di_Pos_Park_Vertical := 3200;
   i_PWM_Cantilever := 1000;
   Rack_Pos[1,1].di_PosRack_Horizontal := 2870;
   Rack_Pos[1,1].di_PosRack_Vertical := 400;
   Rack_Pos[1,2].di_PosRack_Horizontal := 5200;
   Rack_Pos[1,2].di_PosRack_Vertical := 400;
   Rack_Pos[1,3].di_PosRack_Horizontal := 7550;
   Rack_Pos[1,3].di_PosRack_Vertical := 400;
   Rack_Pos[2,1].di_PosRack_Horizontal := 2870;
   Rack_Pos[2,1].di_PosRack_Vertical := 1750;
   Rack_Pos[2,2].di_PosRack_Horizontal := 5200;
   Rack_Pos[2,2].di_PosRack_Vertical := 1750;
   Rack_Pos[2,3].di_PosRack_Horizontal := 7550;
   Rack_Pos[2,3].di_PosRack_Vertical := 1750;
   Rack_Pos[3,1].di_PosRack_Horizontal := 2870;
   Rack_Pos[3,1].di_PosRack_Vertical := 3150;
   Rack_Pos[3,2].di_PosRack_Horizontal := 5200;
   Rack_Pos[3,2].di_PosRack_Vertical := 3150;
   Rack_Pos[3,3].di_PosRack_Horizontal := 7550;
   Rack_Pos[3,3].di_PosRack_Vertical := 3150;
   Rack_Workpiece[1,1].s_id := '0';
   Rack_Workpiece[1,2].s_id := '0';
   Rack_Workpiece[1,3].s_id := '0';
   Rack_Workpiece[2,1].s_id := '0';
   Rack_Workpiece[2,2].s_id := '0';
   Rack_Workpiece[2,3].s_id := '0';
   Rack_Workpiece[3,1].s_id := '0';
   Rack_Workpiece[3,2].s_id := '0';
   Rack_Workpiece[3,3].s_id := '0';
   Horizontal_Axis.i_PWM := 700;
   Horizontal_Axis.Config.di_Pos_Soft_Switch := 7900;
   Horizontal_Axis.Config.di_Pos_Window := 15;
   Vertical_Axis.i_PWM := 600;
   Vertical_Axis.Config.di_Pos_Soft_Switch := 3350;
   Vertical_Axis.Config.di_Pos_Window := 15;
END_DATA_BLOCK

DATA_BLOCK "PRG_HBW_Axis_Horizontal_DB"   // DB18
{ S7_Optimized_Access := 'TRUE' }
AUTHOR : A.Schaefer
VERSION : 0.1
// stored: InstanceOfName PRG_HBW_Axis_Horizontal
"PRG_HBW_Axis_Horizontal"
BEGIN
END_DATA_BLOCK

DATA_BLOCK "PRG_VGR_Ablauf_DB"   // DB19
{ S7_Optimized_Access := 'TRUE' }
AUTHOR : A.Schaefer
VERSION : 0.1
// stored: InstanceOfName PRG_VGR_Ablauf
"PRG_VGR_Ablauf"
BEGIN
END_DATA_BLOCK

DATA_BLOCK "PRG_SLD_Ablauf_DB"   // DB20
{ S7_Optimized_Access := 'TRUE' }
AUTHOR : A.Schaefer
VERSION : 0.1
// stored: InstanceOfName PRG_SLD_Ablauf
"PRG_SLD_Ablauf"
BEGIN
END_DATA_BLOCK

DATA_BLOCK "PRG_Acknowledge_DB"   // DB21
{ S7_Optimized_Access := 'TRUE' }
AUTHOR : A.Schaefer
VERSION : 0.1
// stored: InstanceOfName PRG_Acknowledge
"PRG_Acknowledge"
BEGIN
END_DATA_BLOCK

DATA_BLOCK "PRG_HBW_Ablauf_DB"   // DB22
{ S7_Optimized_Access := 'TRUE' }
AUTHOR : A.Schaefer
VERSION : 0.1
// stored: InstanceOfName PRG_HBW_Ablauf
"PRG_HBW_Ablauf"
BEGIN
END_DATA_BLOCK

DATA_BLOCK "gtyp_Setup"   // DB23
TITLE = Global DB Setup
{ S7_Optimized_Access := 'TRUE' }
AUTHOR : A.Schaefer
VERSION : 0.0
BEGIN
END_DATA_BLOCK

DATA_BLOCK "gtyp_SLD"   // DB24
TITLE = Global DB SLD
{ S7_Optimized_Access := 'TRUE' }
AUTHOR : A.Schaefer
VERSION : 0.0
BEGIN
   i_CounterValue_Blue := 26;
   i_CounterValue_White := 5;
   i_CounterValue_Red := 16;
   w_Threshold_White_Red := 16#2698;
   w_Threshold_Red_Blue := 16#3D41;
END_DATA_BLOCK

DATA_BLOCK "PRG_Order_DB"   // DB25
{ S7_Optimized_Access := 'TRUE' }
AUTHOR : A.Schaefer
VERSION : 0.1
// stored: InstanceOfName PRG_Order
"PRG_Order"
BEGIN
END_DATA_BLOCK

DATA_BLOCK "PRG_SSC_Light_DB"   // DB26
{ S7_Optimized_Access := 'TRUE' }
AUTHOR : A.Schaefer
VERSION : 0.1
// stored: InstanceOfName PRG_SSC_Light
"PRG_SSC_Light"
BEGIN
END_DATA_BLOCK

DATA_BLOCK "PRG_HBW_Axis_Horizontal_Act_Pos_DB"   // DB27
{ S7_Optimized_Access := 'TRUE' }
AUTHOR : A.Schaefer
VERSION : 0.1
// stored: InstanceOfName PRG_HBW_Axis_Horizontal_Act_Pos
"PRG_HBW_Axis_Horizontal_Act_Pos"
BEGIN
END_DATA_BLOCK

DATA_BLOCK "PRG_HBW_Axis_Vertical_Act_Pos_DB"   // DB28
{ S7_Optimized_Access := 'TRUE' }
AUTHOR : A.Schaefer
VERSION : 0.1
// stored: InstanceOfName PRG_HBW_Axis_Vertical_Act_Pos
"PRG_HBW_Axis_Vertical_Act_Pos"
BEGIN
END_DATA_BLOCK

DATA_BLOCK "PRG_VGR_Axis_vertical_Act_Pos_DB"   // DB29
{ S7_Optimized_Access := 'TRUE' }
AUTHOR : A.Schaefer
VERSION : 0.1
// stored: InstanceOfName PRG_VGR_Axis_vertical_Act_Pos
"PRG_VGR_Axis_vertical_Act_Pos"
BEGIN
END_DATA_BLOCK

DATA_BLOCK "PRG_SSC_Axis_Horizontal_Act_Pos_DB"   // DB30
{ S7_Optimized_Access := 'TRUE' }
AUTHOR : A.Schaefer
VERSION : 0.1
// stored: InstanceOfName PRG_SSC_Axis_Horizontal_Act_Pos
"PRG_SSC_Axis_Horizontal_Act_Pos"
BEGIN
END_DATA_BLOCK

DATA_BLOCK "PRG_VGR_Axis_rotate_Act_Pos_DB"   // DB31
{ S7_Optimized_Access := 'TRUE' }
AUTHOR : A.Schaefer
VERSION : 0.1
// stored: InstanceOfName PRG_VGR_Axis_rotate_Act_Pos
"PRG_VGR_Axis_rotate_Act_Pos"
BEGIN
END_DATA_BLOCK

DATA_BLOCK "PRG_DSI_Status_DB"   // DB32
{ S7_Optimized_Access := 'TRUE' }
AUTHOR : A.Schaefer
VERSION : 0.1
// stored: InstanceOfName PRG_DSI_Status
"PRG_DSI_Status"
BEGIN
END_DATA_BLOCK

DATA_BLOCK "PRG_DSO_Status_DB"   // DB33
{ S7_Optimized_Access := 'TRUE' }
AUTHOR : A.Schaefer
VERSION : 0.1
// stored: InstanceOfName PRG_DSO_Status
"PRG_DSO_Status"
BEGIN
END_DATA_BLOCK

DATA_BLOCK "PRG_VGR_Set_Positioning_DB"   // DB34
{ S7_Optimized_Access := 'TRUE' }
AUTHOR : A.Schaefer
VERSION : 0.1
// stored: InstanceOfName PRG_VGR_Set_Positioning
"PRG_VGR_Set_Positioning"
BEGIN
END_DATA_BLOCK

DATA_BLOCK "PRG_HBW_Set_Positioning_DB"   // DB35
{ S7_Optimized_Access := 'TRUE' }
AUTHOR : A.Schaefer
VERSION : 0.1
// stored: InstanceOfName PRG_HBW_Set_Positioning
"PRG_HBW_Set_Positioning"
BEGIN
END_DATA_BLOCK

DATA_BLOCK "PRG_SSC_Set_Positioning_DB"   // DB36
{ S7_Optimized_Access := 'TRUE' }
AUTHOR : A.Schaefer
VERSION : 0.1
// stored: InstanceOfName PRG_SSC_Set_Positioning
"PRG_SSC_Set_Positioning"
BEGIN
END_DATA_BLOCK

DATA_BLOCK "PRG_SSC_Calibration_Color_DB"   // DB37
{ S7_Optimized_Access := 'TRUE' }
AUTHOR : A.Schaefer
VERSION : 0.1
// stored: InstanceOfName PRG_SSC_Calibration_Color
"PRG_SSC_Calibration_Color"
BEGIN
END_DATA_BLOCK

DATA_BLOCK "PRG_SLD_Calibration_Color_DB"   // DB38
{ S7_Optimized_Access := 'TRUE' }
AUTHOR : A.Schaefer
VERSION : 0.1
// stored: InstanceOfName PRG_SLD_Calibration_Color
"PRG_SLD_Calibration_Color"
BEGIN
END_DATA_BLOCK

DATA_BLOCK "PRG_SLD_Set_Counter_Values_DB"   // DB39
{ S7_Optimized_Access := 'TRUE' }
AUTHOR : A.Schaefer
VERSION : 0.1
// stored: InstanceOfName PRG_SLD_Set_Counter_Values
"PRG_SLD_Set_Counter_Values"
BEGIN
END_DATA_BLOCK

DATA_BLOCK "gtyp_Interface_TXT_Controler"   // DB40
{ S7_Optimized_Access := 'TRUE' }
VERSION : 0.1
BEGIN
END_DATA_BLOCK

DATA_BLOCK "PRG_SSC_Set_Park_Position_DB"   // DB41
{ S7_Optimized_Access := 'TRUE' }
AUTHOR : A.Schaefer
VERSION : 0.0
// stored: InstanceOfName PRG_SSC_Set_Park_Position
"PRG_SSC_Set_Park_Position"
BEGIN
END_DATA_BLOCK

DATA_BLOCK "PRG_VGR_Set_Park_Position_DB"   // DB42
{ S7_Optimized_Access := 'TRUE' }
AUTHOR : A.Schaefer
VERSION : 0.0
// stored: InstanceOfName PRG_VGR_Set_Park_Position
"PRG_VGR_Set_Park_Position"
BEGIN
END_DATA_BLOCK

DATA_BLOCK "PRG_HBW_Set_Park_Position_DB"   // DB43
{ S7_Optimized_Access := 'TRUE' }
AUTHOR : A.Schaefer
VERSION : 0.0
// stored: InstanceOfName PRG_HBW_Set_Park_Position
"PRG_HBW_Set_Park_Position"
BEGIN
END_DATA_BLOCK

DATA_BLOCK "PRG_MPO_Set_Park_Position_DB"   // DB44
{ S7_Optimized_Access := 'TRUE' }
AUTHOR : A.Schaefer
VERSION : 0.0
// stored: InstanceOfName PRG_MPO_Set_Park_Position
"PRG_MPO_Set_Park_Position"
BEGIN
END_DATA_BLOCK

DATA_BLOCK "RT_INFO_scl_OB30"   // DB325
{ S7_Optimized_Access := 'TRUE' }
VERSION : 0.1
   VAR
      mode : UInt := 1;   // Mode 1 = Runtime of a specific OB; 2 = Maximum runtime of a specific OB; 3 = Minimum runtime of a specific OB; 10 = Mean value of the percentage of total runtime used by higher-priority OBs; ...
      obNbr : OB_Any := 1;   // OB to read
      infoData : LTime;   // mode 1 --> Runtime in LTIME
      returnValue : Int;   // Error information of instruction
   END_VAR
BEGIN
END_DATA_BLOCK

DATA_BLOCK "RT_INFO_scl_OB1"   // DB326
{ S7_Optimized_Access := 'TRUE' }
VERSION : 0.1
   VAR
      mode : UInt := 1;   // Mode 1 = Runtime of a specific OB; 2 = Maximum runtime of a specific OB; 3 = Minimum runtime of a specific OB; 10 = Mean value of the percentage of total runtime used by higher-priority OBs; ...
      obNbr : OB_Any := 1;   // OB to read
      infoData : LTime;   // mode 1 --> Runtime in LTIME
      returnValue : Int;   // Error information of instruction
   END_VAR
BEGIN
END_DATA_BLOCK

FUNCTION_BLOCK "PRG_VGR_Axis_vertical"   // FB1, SCL
TITLE = Program Axis vertical VGR
{ S7_Optimized_Access := 'TRUE' }
AUTHOR : A.Schaefer
VERSION : 0.0
   VAR
      lx_Init : Bool;
      lfb_vertical_Axis : "FB_Axis";
   END_VAR
BEGIN
   IF #lx_Init THEN

       // FB Axis vertical
       #lfb_vertical_Axis(ini_Axis := 2,
                          indi_Increment := "gtyp_VGR".vertical_Axis.di_Increment,
                          inx_Ref_Switch := "IX_VGR_RefSwitchVerticalAxis_I1",
                          inx_Referencing := "gtyp_VGR".vertical_Axis.x_Reference,
                          inx_Start_Positioning := "gtyp_VGR".vertical_Axis.x_Start_Positioning,
                          indi_Target_Position := "gtyp_VGR".vertical_Axis.di_Target_Position,
                          ini_PWM := "gtyp_VGR".vertical_Axis.i_PWM,
                          inouttyp_Config := "gtyp_VGR".vertical_Axis.Config,
                          inouttyp_Setup := "gtyp_SetupAxis");

       "QX_VGR_M1_VerticalAxisUp_Q1" := #lfb_vertical_Axis.outx_Motor_Neg;
       "QX_VGR_M1_VerticalAxisDown_Q2" := #lfb_vertical_Axis.outx_Motor_Pos;
       "QW_VGR_PWM_Vertical_M1" := #lfb_vertical_Axis.outi_Motor_PWM;
       "gtyp_VGR".vertical_Axis.di_Actual_Position := #lfb_vertical_Axis.outdi_Actual_Position;
       "gtyp_VGR".vertical_Axis.x_Referenced := #lfb_vertical_Axis.outx_Referenced;
       "gtyp_VGR".vertical_Axis.x_Position_Reached := #lfb_vertical_Axis.outx_Position_Reached;
   ELSE
       #lx_Init := TRUE;
   END_IF;
END_FUNCTION_BLOCK

FUNCTION_BLOCK "FB_Blinker"   // FB2, SCL
TITLE = Functionblock Blinker
{ S7_Optimized_Access := 'TRUE' }
AUTHOR : A.Schaefer
VERSION : 0.0
   VAR_INPUT
      int_periodendauer : Time;
   END_VAR
   VAR_OUTPUT
      outx_blinker : Bool;
   END_VAR
   VAR
      lfb_ton : TON_TIME;
      lx_esv_timer : Bool;
      lx_blinker : Bool;
   END_VAR
BEGIN
   #lfb_ton(IN := NOT #lx_esv_timer,
            PT := #int_periodendauer / 2,
            Q => #lx_esv_timer);

   IF #lx_esv_timer THEN
       #lx_blinker := NOT #lx_blinker;
   END_IF;

   #outx_blinker := #lx_blinker;
END_FUNCTION_BLOCK

FUNCTION_BLOCK "PRG_VGR_Axis_horizontal"   // FB4, SCL
TITLE = Program Axis horizontal VGR
{ S7_Optimized_Access := 'TRUE' }
AUTHOR : A.Schaefer
VERSION : 0.0
   VAR
      lx_Init : Bool;
      lfb_horizontal_Axis : "FB_Axis";
   END_VAR
BEGIN
   IF #lx_Init THEN

       // FB Axis horizontal
       #lfb_horizontal_Axis(ini_Axis := 1,
                            indi_Increment := "gtyp_VGR".horizontal_Axis.di_Increment,
                            inx_Ref_Switch := "IX_VGR_RefSwitchHorizontalAxis_I2",
                            inx_Referencing := "gtyp_VGR".horizontal_Axis.x_Reference,
                            inx_Start_Positioning := "gtyp_VGR".horizontal_Axis.x_Start_Positioning,
                            indi_Target_Position := "gtyp_VGR".horizontal_Axis.di_Target_Position,
                            ini_PWM := "gtyp_VGR".horizontal_Axis.i_PWM,
                            inouttyp_Config := "gtyp_VGR".horizontal_Axis.Config,
                            inouttyp_Setup := "gtyp_SetupAxis");

       "QX_VGR_M2_HorizontalAxisForward_Q4" := #lfb_horizontal_Axis.outx_Motor_Pos;
       "QX_VGR_M2_HorizontalAxisBackward_Q3" := #lfb_horizontal_Axis.outx_Motor_Neg;
       "QW_VGR_PWM_Horizontal_M2" := #lfb_horizontal_Axis.outi_Motor_PWM;
       "gtyp_VGR".horizontal_Axis.di_Actual_Position := #lfb_horizontal_Axis.outdi_Actual_Position;
       "gtyp_VGR".horizontal_Axis.x_Referenced := #lfb_horizontal_Axis.outx_Referenced;
       "gtyp_VGR".horizontal_Axis.x_Position_Reached := #lfb_horizontal_Axis.outx_Position_Reached;
   ELSE
       #lx_Init := TRUE;
   END_IF;
END_FUNCTION_BLOCK

FUNCTION_BLOCK "PRG_VGR_Axis_rotate"   // FB5, SCL
TITLE = Program Axis rotate VGR
{ S7_Optimized_Access := 'TRUE' }
AUTHOR : A.Schaefer
VERSION : 0.0
   VAR
      lx_Init : Bool;
      lfb_rotate_Axis : "FB_Axis";
   END_VAR
BEGIN
   IF #lx_Init THEN

       // FB Axis rotate
       #lfb_rotate_Axis(ini_Axis := 3,
                        indi_Increment := "gtyp_VGR".rotate_Axis.di_Increment,
                        inx_Ref_Switch := "IX_VGR_RefSwitchRotate_I3",
                        inx_Referencing := "gtyp_VGR".rotate_Axis.x_Reference,
                        inx_Start_Positioning := "gtyp_VGR".rotate_Axis.x_Start_Positioning,
                        indi_Target_Position := "gtyp_VGR".rotate_Axis.di_Target_Position,
                        ini_PWM := "gtyp_VGR".rotate_Axis.i_PWM,
                        inouttyp_Config := "gtyp_VGR".rotate_Axis.Config,
                        inouttyp_Setup := "gtyp_SetupAxis");

       "QX_VGR_M3_RotateClockwise_Q5" := #lfb_rotate_Axis.outx_Motor_Neg;
       "QX_VGR_M3_RotateCounterclockwise_Q6" := #lfb_rotate_Axis.outx_Motor_Pos;
       "QW_VGR_PWM_Rotate_M3" := #lfb_rotate_Axis.outi_Motor_PWM;
       "gtyp_VGR".rotate_Axis.di_Actual_Position := #lfb_rotate_Axis.outdi_Actual_Position;
       "gtyp_VGR".rotate_Axis.x_Referenced := #lfb_rotate_Axis.outx_Referenced;
       "gtyp_VGR".rotate_Axis.x_Position_Reached := #lfb_rotate_Axis.outx_Position_Reached;
   ELSE
       #lx_Init := TRUE;
   END_IF;
END_FUNCTION_BLOCK

FUNCTION_BLOCK "PRG_VGR_Ablauf"   // FB7, SCL
TITLE = Program Ablauf VGR
{ S7_Optimized_Access := 'TRUE' }
AUTHOR : A.Schaefer
VERSION : 0.0
   VAR
      lx_Init : Bool;
      lx_Start_TON_Wait : Bool;
      lx_Start_TON_State : Bool;
      lt_TON_Wait : Time;
      ldt_MQTT : Date_And_Time;
      li_Return_LDT : Int;
      li_Lights : Int;
      li_Lights_old : Int;
      lx_State_activ : Bool;
      li_StepCase : Int;
      li_Counter : Int;
      ldi_Pos_SLD_X : DInt;
      ldi_Pos_SLD_Y : DInt;
      ldi_Pos_SLD_Z : DInt;
      ls_Color : String;
      ls_Target : String;
      lfb_TON_Wait : TON_TIME;
      lfb_TON_State : TON_TIME;
      lfb_R_Trig_NiO : R_TRIG;
   END_VAR
BEGIN
   IF #lx_Init THEN

       // Restart after set Positioning
       IF "gtyp_Setup".x_Set_Pos_Activ OR "gtyp_Setup".x_Color_Sensor_Calibration OR "gtyp_VGR".x_Start_Park_Position OR "gtyp_MPO".x_Error THEN
           IF "gtyp_MPO".x_Error THEN
               "gtyp_VGR".x_MPO_Req_Discard := FALSE;
               "gtyp_VGR".x_MPO_Discards := FALSE;
           END_IF;
           #li_StepCase := 0;
       END_IF;

       // wait time state
       #lfb_TON_State(IN := NOT #lx_Start_TON_State,
                      PT := T#2s);

       IF "gtyp_VGR".x_State_Process THEN
           #li_Return_LDT := RD_SYS_T(#ldt_MQTT);
           "gtyp_Interface_Dashboard".Subscribe.State_Order.ldt_ts := DT_TO_LDT(#ldt_MQTT);
       END_IF;

       // state of the robot cyclically transmitted to the cloud
       IF (#lfb_TON_State.Q OR (#li_Lights <> #li_Lights_old)) AND NOT #lx_Start_TON_State THEN
           #li_Lights_old := #li_Lights;
           #lx_Start_TON_State := TRUE;
           #li_Return_LDT := RD_SYS_T(#ldt_MQTT);
           "gtyp_Interface_Dashboard".Subscribe.State_VGR.ldt_ts := DT_TO_LDT(#ldt_MQTT);
           "gtyp_Interface_Dashboard".Subscribe.State_VGR.i_code := #li_Lights;
           "gtyp_Interface_Dashboard".Subscribe.State_VGR.s_description := '';
           "gtyp_Interface_Dashboard".Subscribe.State_VGR.s_station := 'vgr';
           "gtyp_Interface_Dashboard".Subscribe.State_VGR.s_target := #ls_Target;
           "gtyp_Interface_Dashboard".Subscribe.State_VGR.x_active := #lx_State_activ;

           "gtyp_Interface_Dashboard".Subscribe.PosPanTiltUnit.ldt_ts := DT_TO_LDT(#ldt_MQTT);
       END_IF;

       // restart wait time state
       IF NOT #lfb_TON_State.Q AND #lx_Start_TON_State THEN
           #lx_Start_TON_State := FALSE;
       END_IF;

       // rising edge Workpiece NiO
       #lfb_R_Trig_NiO(CLK := "gtyp_VGR".x_Workpiece_NiO);

       IF #lfb_R_Trig_NiO.Q THEN
           #lx_Start_TON_Wait := FALSE;
           #lx_State_activ := FALSE;
           #li_Lights := 4;
           #ls_Target := '';
           "gtyp_VGR".horizontal_Axis.x_Start_Positioning := FALSE;
           "gtyp_VGR".vertical_Axis.x_Start_Positioning := FALSE;
           "gtyp_VGR".rotate_Axis.x_Start_Positioning := FALSE;
           "gtyp_VGR".x_NFC_Start_First := FALSE;
           "gtyp_VGR".x_NFC_Start := FALSE;
           #li_StepCase := 70;
       END_IF;

       // FB TON Wait
       #lfb_TON_Wait(IN := #lx_Start_TON_Wait,
                     PT := #lt_TON_Wait);

       // step chain VGR
       CASE #li_StepCase OF

           0:  // init
               #lx_Start_TON_Wait := FALSE;
               #li_Lights := 1;
               #lx_State_activ := FALSE;
               #ls_Target := '';
               "gtyp_VGR".horizontal_Axis.x_Start_Positioning := FALSE;
               "gtyp_VGR".vertical_Axis.x_Start_Positioning := FALSE;
               "gtyp_VGR".rotate_Axis.x_Start_Positioning := FALSE;
               "gtyp_VGR".x_HBW_Storage := FALSE;
               "gtyp_VGR".x_HBW_Outsource := FALSE;
               "gtyp_VGR".x_NFC_Start_First := FALSE;
               "gtyp_VGR".x_NFC_Start := FALSE;
               "gtyp_VGR".x_Ready_For_Outsource := FALSE;
               "QX_VGR_Compressor_Q7" := FALSE;
               "QX_VGR_ValveVacuum_Q8" := FALSE;

               IF NOT "gtyp_Setup".x_Set_Pos_Activ AND NOT "gtyp_VGR".x_Start_Park_Position AND NOT "gtyp_MPO".x_Error THEN
                   #li_StepCase := 10;
               END_IF;

           10: // homing vertical axis
               #li_Lights := 2;
               "gtyp_VGR".x_Ready_For_Outsource := TRUE;
               "gtyp_VGR".vertical_Axis.x_Reference := TRUE;
               "gtyp_VGR".vertical_Axis.i_PWM := 800;

               IF NOT "gtyp_VGR".vertical_Axis.x_Referenced THEN
                   #li_StepCase := 20;
               END_IF;

           20: // homed vertical axis
               IF "gtyp_VGR".vertical_Axis.x_Referenced THEN
                   "gtyp_VGR".vertical_Axis.x_Reference := FALSE;
                   #li_StepCase := 30;
               END_IF;

           30: // homing horizontal axis
               "gtyp_VGR".horizontal_Axis.x_Reference := TRUE;

               IF NOT "gtyp_VGR".horizontal_Axis.x_Referenced THEN
                   #li_StepCase := 40;
               END_IF;

           40: // homed horizontal axis
               IF "gtyp_VGR".horizontal_Axis.x_Referenced THEN
                   "gtyp_VGR".horizontal_Axis.x_Reference := FALSE;
                   #li_StepCase := 50;
               END_IF;

           50: // homing rotate axis
               "gtyp_VGR".rotate_Axis.x_Reference := TRUE;

               IF NOT "gtyp_VGR".rotate_Axis.x_Referenced THEN
                   #li_StepCase := 60;
               END_IF;

           60: // homed rotate axis
               IF "gtyp_VGR".rotate_Axis.x_Referenced THEN
                   "gtyp_VGR".rotate_Axis.x_Reference := FALSE;
                   #li_StepCase := 70;
               END_IF;

           70: // Deciding which route to take

               #li_Lights := 1;
               #lx_State_activ := FALSE;
               #ls_Target := '';
               "gtyp_VGR".x_Ready_For_Outsource := TRUE;

               // Procedure - bad part
               IF "gtyp_VGR".x_Workpiece_NiO THEN
                   "gtyp_VGR".x_Ready_For_Outsource := FALSE;
                   #li_Lights := 4;
                   #li_StepCase := 1200;
                   // Procedure - pick up finished parts blue
               ELSIF NOT "IX_SLD_LightBarrierBlue_I7" THEN
                   #ldi_Pos_SLD_X := "gtyp_VGR".di_Pos_SLD_Blue_horizontal;
                   #ldi_Pos_SLD_Y := "gtyp_VGR".di_Pos_SLD_Blue_vertical;
                   #ldi_Pos_SLD_Z := "gtyp_VGR".di_Pos_SLD_Blue_rotate;
                   "gtyp_VGR".x_Ready_For_Outsource := FALSE;
                   #li_StepCase := 100;
                   // Procedure - pick up finished parts red
               ELSIF NOT "IX_SLD_LightBarrierRed_I6" THEN
                   #ldi_Pos_SLD_X := "gtyp_VGR".di_Pos_SLD_Red_horizontal;
                   #ldi_Pos_SLD_Y := "gtyp_VGR".di_Pos_SLD_Red_vertical;
                   #ldi_Pos_SLD_Z := "gtyp_VGR".di_Pos_SLD_Red_rotate;
                   "gtyp_VGR".x_Ready_For_Outsource := FALSE;
                   #li_StepCase := 100;
                   // Procedure - pick up finished parts white
               ELSIF NOT "IX_SLD_LightBarrierWhite_I5" THEN
                   #ldi_Pos_SLD_X := "gtyp_VGR".di_Pos_SLD_White_horizontal;
                   #ldi_Pos_SLD_Y := "gtyp_VGR".di_Pos_SLD_White_vertical;
                   #ldi_Pos_SLD_Z := "gtyp_VGR".di_Pos_SLD_White_rotate;
                   "gtyp_VGR".x_Ready_For_Outsource := FALSE;
                   #li_StepCase := 100;
                   // Procedure - outsource to manufacturing
               ELSIF "gtyp_VGR".x_HBW_Outsource THEN
                   // Order State
                   "gtyp_Interface_Dashboard".Subscribe.State_Order.ldt_ts := DT_TO_LDT(#ldt_MQTT);
                   "gtyp_Interface_Dashboard".Subscribe.State_Order.s_state := 'ORDERED';
                   "gtyp_Interface_Dashboard".Subscribe.State_Order.s_type := "gtyp_VGR".s_HBW_Outsource_Typ;
                   #li_StepCase := 400;
                   // Procedure - store raw parts
               ELSIF NOT "IX_SSC_LightBarrierStorage_I3" THEN
                   "gtyp_VGR".x_Ready_For_Outsource := FALSE;
                   #li_Lights := 2;
                   "gtyp_VGR".x_HBW_Storage := TRUE;
                   #li_StepCase := 600;
               END_IF;

               (**************************************************************************************************)
               (****************************    Procedure - pick up finished parts    ****************************)
               (**************************************************************************************************)
           100: // Position of finished part 

               #li_Lights := 2;
               "gtyp_VGR".horizontal_Axis.di_Target_Position := #ldi_Pos_SLD_X;
               "gtyp_VGR".horizontal_Axis.x_Start_Positioning := TRUE;

               "gtyp_VGR".vertical_Axis.x_Reference := TRUE;
               "gtyp_VGR".vertical_Axis.i_PWM := 800;

               "gtyp_VGR".rotate_Axis.di_Target_Position := #ldi_Pos_SLD_Z;
               "gtyp_VGR".rotate_Axis.x_Start_Positioning := TRUE;

               IF ("gtyp_VGR".horizontal_Axis.di_Actual_Position <= (#ldi_Pos_SLD_X + "gtyp_VGR".horizontal_Axis.Config.di_Pos_Window))
                   AND ("gtyp_VGR".horizontal_Axis.di_Actual_Position >= (#ldi_Pos_SLD_X - "gtyp_VGR".horizontal_Axis.Config.di_Pos_Window))
                   AND "gtyp_VGR".horizontal_Axis.x_Position_Reached THEN
                   "gtyp_VGR".horizontal_Axis.x_Start_Positioning := FALSE;
               END_IF;

               IF ("gtyp_VGR".rotate_Axis.di_Actual_Position <= (#ldi_Pos_SLD_Z + "gtyp_VGR".rotate_Axis.Config.di_Pos_Window))
                   AND ("gtyp_VGR".rotate_Axis.di_Actual_Position >= (#ldi_Pos_SLD_Z - "gtyp_VGR".rotate_Axis.Config.di_Pos_Window))
                   AND "gtyp_VGR".rotate_Axis.x_Position_Reached THEN
                   "gtyp_VGR".rotate_Axis.x_Start_Positioning := FALSE;
               END_IF;

               IF NOT "gtyp_VGR".vertical_Axis.x_Referenced THEN
                   #li_StepCase := 110;
               END_IF;

           110: // position of finished part reached         

               IF ("gtyp_VGR".horizontal_Axis.di_Actual_Position <= (#ldi_Pos_SLD_X + "gtyp_VGR".horizontal_Axis.Config.di_Pos_Window))
                   AND ("gtyp_VGR".horizontal_Axis.di_Actual_Position >= (#ldi_Pos_SLD_X - "gtyp_VGR".horizontal_Axis.Config.di_Pos_Window))
                   AND "gtyp_VGR".horizontal_Axis.x_Position_Reached THEN
                   "gtyp_VGR".horizontal_Axis.x_Start_Positioning := FALSE;
               END_IF;

               IF ("gtyp_VGR".rotate_Axis.di_Actual_Position <= (#ldi_Pos_SLD_Z + "gtyp_VGR".rotate_Axis.Config.di_Pos_Window))
                   AND ("gtyp_VGR".rotate_Axis.di_Actual_Position >= (#ldi_Pos_SLD_Z - "gtyp_VGR".rotate_Axis.Config.di_Pos_Window))
                   AND "gtyp_VGR".rotate_Axis.x_Position_Reached THEN
                   "gtyp_VGR".rotate_Axis.x_Start_Positioning := FALSE;
               END_IF;

               IF "gtyp_VGR".vertical_Axis.x_Referenced THEN
                   "gtyp_VGR".vertical_Axis.x_Reference := FALSE;
               END_IF;

               IF ("gtyp_VGR".horizontal_Axis.di_Actual_Position <= (#ldi_Pos_SLD_X + "gtyp_VGR".horizontal_Axis.Config.di_Pos_Window))
                   AND ("gtyp_VGR".horizontal_Axis.di_Actual_Position >= (#ldi_Pos_SLD_X - "gtyp_VGR".horizontal_Axis.Config.di_Pos_Window))
                   AND "gtyp_VGR".horizontal_Axis.x_Position_Reached
                   AND "gtyp_VGR".vertical_Axis.x_Referenced
                   AND ("gtyp_VGR".rotate_Axis.di_Actual_Position <= (#ldi_Pos_SLD_Z + "gtyp_VGR".rotate_Axis.Config.di_Pos_Window))
                   AND ("gtyp_VGR".rotate_Axis.di_Actual_Position >= (#ldi_Pos_SLD_Z - "gtyp_VGR".rotate_Axis.Config.di_Pos_Window))
                   AND "gtyp_VGR".rotate_Axis.x_Position_Reached THEN
                   "gtyp_VGR".horizontal_Axis.x_Start_Positioning := FALSE;
                   "gtyp_VGR".vertical_Axis.x_Start_Positioning := FALSE;
                   "gtyp_VGR".rotate_Axis.x_Start_Positioning := FALSE;
                   #li_StepCase := 120;
               END_IF;

           120: // wait sequence
               #lx_Start_TON_Wait := TRUE;
               #lt_TON_Wait := T#500ms;

               IF #lfb_TON_Wait.Q THEN
                   #lx_Start_TON_Wait := FALSE;
                   #li_StepCase := 130;
               END_IF;

           130: // Position vertical finished part
               "gtyp_VGR".vertical_Axis.di_Target_Position := #ldi_Pos_SLD_Y;
               "gtyp_VGR".vertical_Axis.x_Start_Positioning := TRUE;
               "gtyp_VGR".vertical_Axis.i_PWM := 500;

               IF ("gtyp_VGR".vertical_Axis.di_Actual_Position <= (#ldi_Pos_SLD_Y + "gtyp_VGR".vertical_Axis.Config.di_Pos_Window))
                   AND ("gtyp_VGR".vertical_Axis.di_Actual_Position >= (#ldi_Pos_SLD_Y - "gtyp_VGR".vertical_Axis.Config.di_Pos_Window))
                   AND "gtyp_VGR".vertical_Axis.x_Position_Reached THEN
                   "gtyp_VGR".vertical_Axis.x_Start_Positioning := FALSE;
                   #li_StepCase := 140;
               END_IF;

           140: // start compressor
               "QX_VGR_Compressor_Q7" := TRUE;

               #lx_Start_TON_Wait := TRUE;
               #lt_TON_Wait := T#1000ms;

               IF #lfb_TON_Wait.Q THEN
                   #lx_Start_TON_Wait := FALSE;
                   #li_StepCase := 150;
               END_IF;

           150: // turn on the vacuum and pick up the part
               "QX_VGR_ValveVacuum_Q8" := true;

               #lx_Start_TON_Wait := TRUE;
               #lt_TON_Wait := T#1000ms;

               IF #lfb_TON_Wait.Q THEN
                   #lx_Start_TON_Wait := FALSE;
                   #lx_State_activ := TRUE;
                   #ls_Target := 'dso';
                   "gtyp_VGR".History := "gtyp_SLD".History;
                   "gtyp_VGR".Workpiece := "gtyp_SLD".Workpiece;
                   "gtyp_SLD".Workpiece.s_id := '0';
                   "gtyp_SLD".Workpiece.s_state := '';
                   "gtyp_SLD".Workpiece.s_type := '';
                   FOR #li_Counter := 1 TO 8 DO
                       "gtyp_SLD".History[#li_Counter].i_code := 0;
                       "gtyp_SLD".History[#li_Counter].ldt_ts := DT#1990-01-01-00:00:00;
                   END_FOR;

                   #li_Return_LDT := RD_SYS_T(#ldt_MQTT);
                   "gtyp_VGR".History[8].i_code := 800;
                   "gtyp_VGR".History[8].ldt_ts := DT_TO_LDT(#ldt_MQTT);

                   "gtyp_Interface_Dashboard".Subscribe.State_SLD.x_active := FALSE;

                   #li_StepCase := 160;
               END_IF;

           160: // Position vertical preposition NFC
               "gtyp_VGR".vertical_Axis.di_Target_Position := "gtyp_VGR".di_Pos_NFC_vertical - "gtyp_VGR".di_Offset_Pos_DSI_NFC_vertical;
               "gtyp_VGR".vertical_Axis.x_Start_Positioning := TRUE;
               "gtyp_VGR".vertical_Axis.i_PWM := 800;

               IF ("gtyp_VGR".vertical_Axis.di_Actual_Position <= ("gtyp_VGR".di_Pos_NFC_vertical - "gtyp_VGR".di_Offset_Pos_DSI_NFC_vertical + "gtyp_VGR".vertical_Axis.Config.di_Pos_Window))
                   AND ("gtyp_VGR".vertical_Axis.di_Actual_Position >= ("gtyp_VGR".di_Pos_NFC_vertical - "gtyp_VGR".di_Offset_Pos_DSI_NFC_vertical - "gtyp_VGR".vertical_Axis.Config.di_Pos_Window))
                   AND "gtyp_VGR".vertical_Axis.x_Position_Reached THEN
                   "gtyp_VGR".vertical_Axis.x_Start_Positioning := FALSE;
                   #li_StepCase := 170;
               END_IF;

           170: // homing horizontal axis
               "gtyp_VGR".horizontal_Axis.x_Reference := TRUE;

               IF NOT "gtyp_VGR".horizontal_Axis.x_Referenced THEN
                   #li_StepCase := 180;
               END_IF;

           180: // homed horizontal axis
               IF "gtyp_VGR".horizontal_Axis.x_Referenced THEN
                   "gtyp_VGR".horizontal_Axis.x_Reference := FALSE;
                   #li_StepCase := 190;
               END_IF;

           190: // wait sequence
               #lx_Start_TON_Wait := TRUE;
               #lt_TON_Wait := T#500ms;

               IF #lfb_TON_Wait.Q THEN
                   #lx_Start_TON_Wait := FALSE;
                   #li_StepCase := 200;
               END_IF;

           200: // Position horizontal/rotate NFC

               "gtyp_VGR".horizontal_Axis.di_Target_Position := "gtyp_VGR".di_Pos_NFC_horizontal;
               "gtyp_VGR".horizontal_Axis.x_Start_Positioning := TRUE;
               "gtyp_VGR".rotate_Axis.di_Target_Position := "gtyp_VGR".di_Pos_NFC_rotate;
               "gtyp_VGR".rotate_Axis.x_Start_Positioning := TRUE;

               IF ("gtyp_VGR".horizontal_Axis.di_Actual_Position <= ("gtyp_VGR".di_Pos_NFC_horizontal + "gtyp_VGR".horizontal_Axis.Config.di_Pos_Window))
                   AND ("gtyp_VGR".horizontal_Axis.di_Actual_Position >= ("gtyp_VGR".di_Pos_NFC_horizontal - "gtyp_VGR".horizontal_Axis.Config.di_Pos_Window))
                   AND "gtyp_VGR".horizontal_Axis.x_Position_Reached THEN
                   "gtyp_VGR".horizontal_Axis.x_Start_Positioning := FALSE;
               END_IF;

               IF ("gtyp_VGR".rotate_Axis.di_Actual_Position <= ("gtyp_VGR".di_Pos_NFC_rotate + "gtyp_VGR".rotate_Axis.Config.di_Pos_Window))
                   AND ("gtyp_VGR".rotate_Axis.di_Actual_Position >= ("gtyp_VGR".di_Pos_NFC_rotate - "gtyp_VGR".rotate_Axis.Config.di_Pos_Window))
                   AND "gtyp_VGR".rotate_Axis.x_Position_Reached THEN
                   "gtyp_VGR".rotate_Axis.x_Start_Positioning := FALSE;
               END_IF;

               IF ("gtyp_VGR".horizontal_Axis.di_Actual_Position <= ("gtyp_VGR".di_Pos_NFC_horizontal + "gtyp_VGR".horizontal_Axis.Config.di_Pos_Window))
                   AND ("gtyp_VGR".horizontal_Axis.di_Actual_Position >= ("gtyp_VGR".di_Pos_NFC_horizontal - "gtyp_VGR".horizontal_Axis.Config.di_Pos_Window))
                   AND "gtyp_VGR".horizontal_Axis.x_Position_Reached
                   AND ("gtyp_VGR".rotate_Axis.di_Actual_Position <= ("gtyp_VGR".di_Pos_NFC_rotate + "gtyp_VGR".rotate_Axis.Config.di_Pos_Window))
                   AND ("gtyp_VGR".rotate_Axis.di_Actual_Position >= ("gtyp_VGR".di_Pos_NFC_rotate - "gtyp_VGR".rotate_Axis.Config.di_Pos_Window))
                   AND "gtyp_VGR".rotate_Axis.x_Position_Reached THEN
                   "gtyp_VGR".horizontal_Axis.x_Start_Positioning := FALSE;
                   "gtyp_VGR".rotate_Axis.x_Start_Positioning := FALSE;
                   #li_StepCase := 210;
               END_IF;

           210: // wait sequence
               #lx_Start_TON_Wait := TRUE;
               #lt_TON_Wait := T#500ms;

               IF #lfb_TON_Wait.Q THEN
                   #lx_Start_TON_Wait := FALSE;
                   #li_StepCase := 220;
               END_IF;

           220: // Position vertical NFC

               "gtyp_VGR".vertical_Axis.di_Target_Position := "gtyp_VGR".di_Pos_NFC_vertical;
               "gtyp_VGR".vertical_Axis.x_Start_Positioning := TRUE;
               "gtyp_VGR".vertical_Axis.i_PWM := 500;

               IF ("gtyp_VGR".vertical_Axis.di_Actual_Position <= ("gtyp_VGR".di_Pos_NFC_vertical + "gtyp_VGR".vertical_Axis.Config.di_Pos_Window))
                   AND ("gtyp_VGR".vertical_Axis.di_Actual_Position >= ("gtyp_VGR".di_Pos_NFC_vertical - "gtyp_VGR".vertical_Axis.Config.di_Pos_Window))
                   AND "gtyp_VGR".vertical_Axis.x_Position_Reached THEN
                   "gtyp_VGR".vertical_Axis.x_Start_Positioning := FALSE;
                   #li_StepCase := 230;
               END_IF;

           230: // Start write/read NFC

               "gtyp_VGR".x_NFC_Start := TRUE;

               IF "gtyp_VGR".x_NFC_Completed THEN
                   "gtyp_VGR".x_NFC_Start := FALSE;
                   #li_StepCase := 240;
               END_IF;

           240: // homing vertical axis

               "gtyp_VGR".vertical_Axis.x_Reference := TRUE;
               "gtyp_VGR".vertical_Axis.i_PWM := 800;

               IF NOT "gtyp_VGR".vertical_Axis.x_Referenced THEN
                   #li_StepCase := 250;
               END_IF;

           250: // homed vertical axis
               IF "gtyp_VGR".vertical_Axis.x_Referenced THEN
                   "gtyp_VGR".vertical_Axis.x_Reference := FALSE;
                   #li_StepCase := 260;
               END_IF;

           260: // wait sequence
               #lx_Start_TON_Wait := TRUE;
               #lt_TON_Wait := T#500ms;

               IF #lfb_TON_Wait.Q THEN
                   #lx_Start_TON_Wait := FALSE;
                   #li_StepCase := 270;
               END_IF;

           270: // Position horizontal/rotate DSO Output

               "gtyp_VGR".horizontal_Axis.di_Target_Position := "gtyp_VGR".di_Pos_DSO_horizontal;
               "gtyp_VGR".horizontal_Axis.x_Start_Positioning := TRUE;

               "gtyp_VGR".rotate_Axis.di_Target_Position := "gtyp_VGR".di_Pos_DSO_rotate;
               "gtyp_VGR".rotate_Axis.x_Start_Positioning := TRUE;

               IF ("gtyp_VGR".horizontal_Axis.di_Actual_Position <= ("gtyp_VGR".di_Pos_DSO_horizontal + "gtyp_VGR".horizontal_Axis.Config.di_Pos_Window))
                   AND ("gtyp_VGR".horizontal_Axis.di_Actual_Position >= ("gtyp_VGR".di_Pos_DSO_horizontal - "gtyp_VGR".horizontal_Axis.Config.di_Pos_Window))
                   AND "gtyp_VGR".horizontal_Axis.x_Position_Reached THEN
                   "gtyp_VGR".horizontal_Axis.x_Start_Positioning := FALSE;
               END_IF;

               IF ("gtyp_VGR".rotate_Axis.di_Actual_Position <= ("gtyp_VGR".di_Pos_DSO_rotate + "gtyp_VGR".rotate_Axis.Config.di_Pos_Window))
                   AND ("gtyp_VGR".rotate_Axis.di_Actual_Position >= ("gtyp_VGR".di_Pos_DSO_rotate - "gtyp_VGR".rotate_Axis.Config.di_Pos_Window))
                   AND "gtyp_VGR".rotate_Axis.x_Position_Reached THEN
                   "gtyp_VGR".rotate_Axis.x_Start_Positioning := FALSE;
               END_IF;
               IF ("gtyp_VGR".horizontal_Axis.di_Actual_Position <= ("gtyp_VGR".di_Pos_DSO_horizontal + "gtyp_VGR".horizontal_Axis.Config.di_Pos_Window))
                   AND ("gtyp_VGR".horizontal_Axis.di_Actual_Position >= ("gtyp_VGR".di_Pos_DSO_horizontal - "gtyp_VGR".horizontal_Axis.Config.di_Pos_Window))
                   AND "gtyp_VGR".horizontal_Axis.x_Position_Reached
                   AND ("gtyp_VGR".rotate_Axis.di_Actual_Position <= ("gtyp_VGR".di_Pos_DSO_rotate + "gtyp_VGR".rotate_Axis.Config.di_Pos_Window))
                   AND ("gtyp_VGR".rotate_Axis.di_Actual_Position >= ("gtyp_VGR".di_Pos_DSO_rotate - "gtyp_VGR".rotate_Axis.Config.di_Pos_Window))
                   AND "gtyp_VGR".rotate_Axis.x_Position_Reached
                   AND "IX_SSC_LightBarrierOutsourcing_I4" THEN
                   "gtyp_VGR".horizontal_Axis.x_Start_Positioning := FALSE;
                   "gtyp_VGR".rotate_Axis.x_Start_Positioning := FALSE;
                   #li_StepCase := 280;
               END_IF;

           280: // Position vertical DSO discard output

               "gtyp_VGR".vertical_Axis.di_Target_Position := "gtyp_VGR".di_Pos_DSO_Discard_vertical;
               "gtyp_VGR".vertical_Axis.x_Start_Positioning := TRUE;
               "gtyp_VGR".vertical_Axis.i_PWM := 500;

               IF ("gtyp_VGR".vertical_Axis.di_Actual_Position <= ("gtyp_VGR".di_Pos_DSO_Discard_vertical + "gtyp_VGR".vertical_Axis.Config.di_Pos_Window))
                   AND ("gtyp_VGR".vertical_Axis.di_Actual_Position >= ("gtyp_VGR".di_Pos_DSO_Discard_vertical - "gtyp_VGR".vertical_Axis.Config.di_Pos_Window))
                   AND "gtyp_VGR".vertical_Axis.x_Position_Reached THEN
                   "gtyp_VGR".vertical_Axis.x_Start_Positioning := FALSE;
                   "gtyp_VGR".x_State_Process := FALSE;
                   "gtyp_VGR".vertical_Axis.i_PWM := 800;
                   #li_StepCase := 290;
               END_IF;

           290: // turn off vacuum
               "QX_VGR_ValveVacuum_Q8" := FALSE;

               #lx_Start_TON_Wait := TRUE;
               #lt_TON_Wait := T#500ms;

               IF #lfb_TON_Wait.Q THEN
                   #li_Return_LDT := RD_SYS_T(#ldt_MQTT);
                   // Order State
                   "gtyp_Interface_Dashboard".Subscribe.State_Order.ldt_ts := DT_TO_LDT(#ldt_MQTT);
                   "gtyp_Interface_Dashboard".Subscribe.State_Order.s_state := 'SHIPPED';
                   "gtyp_Interface_Dashboard".Subscribe.State_Order.s_type := "gtyp_VGR".Workpiece.s_type;
                   "gtyp_SSC".Workpiece := "gtyp_VGR".Workpiece;
                   "gtyp_SSC".History := "gtyp_VGR".History;
                   "gtyp_VGR".Workpiece.s_id := '0';
                   "gtyp_VGR".Workpiece.s_state := '';
                   "gtyp_VGR".Workpiece.s_type := '';
                   FOR #li_Counter := 1 TO 8 DO
                       "gtyp_VGR".History[#li_Counter].i_code := 0;
                       "gtyp_VGR".History[#li_Counter].ldt_ts := DT#1990-01-01-00:00:00;
                   END_FOR;

                   "gtyp_Interface_Dashboard".Subscribe.State_DSO.x_active := TRUE;

                   #lx_Start_TON_Wait := FALSE;
                   #li_StepCase := 300;
               END_IF;

           300: // turn off compressor
               "QX_VGR_Compressor_Q7" := FALSE;
               #lx_State_activ := FALSE;
               #ls_Target := '';
               #li_StepCase := 310;

           310: // homing vertical axis
               "gtyp_VGR".vertical_Axis.x_Reference := TRUE;

               IF NOT "gtyp_VGR".vertical_Axis.x_Referenced THEN
                   #li_StepCase := 320;
               END_IF;

           320: // homed vertical axis
               IF "gtyp_VGR".vertical_Axis.x_Referenced THEN
                   "gtyp_VGR".vertical_Axis.x_Reference := FALSE;
                   #li_StepCase := 330;
               END_IF;

           330: // homing horizontal/rotate axis
               "gtyp_VGR".horizontal_Axis.x_Reference := TRUE;
               "gtyp_VGR".rotate_Axis.x_Reference := TRUE;

               IF NOT "gtyp_VGR".horizontal_Axis.x_Referenced AND NOT "gtyp_VGR".rotate_Axis.x_Referenced THEN
                   #li_StepCase := 340;
               END_IF;

           340: // homed horizontal/rotate axis
               IF "gtyp_VGR".horizontal_Axis.x_Referenced AND "gtyp_VGR".rotate_Axis.x_Referenced THEN
                   "gtyp_VGR".horizontal_Axis.x_Reference := FALSE;
                   "gtyp_VGR".rotate_Axis.x_Reference := FALSE;
                   #li_StepCase := 350;
               END_IF;

           350: // wait sequence
               #lx_Start_TON_Wait := TRUE;
               #lt_TON_Wait := T#500ms;

               IF #lfb_TON_Wait.Q THEN
                   #lx_Start_TON_Wait := FALSE;
                   #li_StepCase := 70;
               END_IF;

               (*******************************************************************************************)
               (****************************           outsource HBW           ****************************)
               (*******************************************************************************************)
           400: // Position rotate HBW and homing vertical/horizontal axis
               #li_Lights := 2;
               "gtyp_VGR".rotate_Axis.di_Target_Position := "gtyp_VGR".di_Pos_HBW_rotate;
               "gtyp_VGR".rotate_Axis.x_Start_Positioning := TRUE;

               "gtyp_VGR".horizontal_Axis.x_Reference := TRUE;
               "gtyp_VGR".vertical_Axis.x_Reference := TRUE;

               IF ("gtyp_VGR".rotate_Axis.di_Actual_Position <= ("gtyp_VGR".di_Pos_HBW_rotate + "gtyp_VGR".rotate_Axis.Config.di_Pos_Window))
                   AND ("gtyp_VGR".rotate_Axis.di_Actual_Position >= ("gtyp_VGR".di_Pos_HBW_rotate - "gtyp_VGR".rotate_Axis.Config.di_Pos_Window))
                   AND "gtyp_VGR".rotate_Axis.x_Position_Reached THEN
                   "gtyp_VGR".rotate_Axis.x_Start_Positioning := FALSE;
               END_IF;

               IF NOT "gtyp_VGR".horizontal_Axis.x_Referenced AND NOT "gtyp_VGR".vertical_Axis.x_Referenced THEN
                   #li_StepCase := 410;
               END_IF;

           410: // Position reached rotate HBW and homed vertical/horizontal axis

               IF ("gtyp_VGR".rotate_Axis.di_Actual_Position <= ("gtyp_VGR".di_Pos_HBW_rotate + "gtyp_VGR".rotate_Axis.Config.di_Pos_Window))
                   AND ("gtyp_VGR".rotate_Axis.di_Actual_Position >= ("gtyp_VGR".di_Pos_HBW_rotate - "gtyp_VGR".rotate_Axis.Config.di_Pos_Window))
                   AND "gtyp_VGR".rotate_Axis.x_Position_Reached THEN
                   "gtyp_VGR".rotate_Axis.x_Start_Positioning := FALSE;
               END_IF;

               IF "gtyp_VGR".horizontal_Axis.x_Referenced THEN
                   "gtyp_VGR".horizontal_Axis.x_Reference := FALSE;
               END_IF;
               IF "gtyp_VGR".vertical_Axis.x_Referenced THEN
                   "gtyp_VGR".vertical_Axis.x_Reference := FALSE;
               END_IF;
               IF "gtyp_VGR".horizontal_Axis.x_Referenced
                   AND "gtyp_VGR".vertical_Axis.x_Referenced
                   AND ("gtyp_VGR".rotate_Axis.di_Actual_Position <= ("gtyp_VGR".di_Pos_HBW_rotate + "gtyp_VGR".rotate_Axis.Config.di_Pos_Window))
                   AND ("gtyp_VGR".rotate_Axis.di_Actual_Position >= ("gtyp_VGR".di_Pos_HBW_rotate - "gtyp_VGR".rotate_Axis.Config.di_Pos_Window))
                   AND "gtyp_VGR".rotate_Axis.x_Position_Reached THEN
                   "gtyp_VGR".horizontal_Axis.x_Reference := FALSE;
                   "gtyp_VGR".vertical_Axis.x_Reference := FALSE;
                   "gtyp_VGR".rotate_Axis.x_Start_Positioning := FALSE;
                   #li_StepCase := 420;
               END_IF;

           420: // wait sequence
               #lx_Start_TON_Wait := TRUE;
               #lt_TON_Wait := T#500ms;

               IF #lfb_TON_Wait.Q THEN
                   #lx_Start_TON_Wait := FALSE;
                   #li_StepCase := 430;
               END_IF;

           430: // Position horizontal HBW 

               "gtyp_VGR".horizontal_Axis.di_Target_Position := "gtyp_VGR".di_Pos_HBW_horizontal;
               "gtyp_VGR".horizontal_Axis.x_Start_Positioning := TRUE;

               IF ("gtyp_VGR".horizontal_Axis.di_Actual_Position <= ("gtyp_VGR".di_Pos_HBW_horizontal + "gtyp_VGR".horizontal_Axis.Config.di_Pos_Window))
                   AND ("gtyp_VGR".horizontal_Axis.di_Actual_Position >= ("gtyp_VGR".di_Pos_HBW_horizontal - "gtyp_VGR".horizontal_Axis.Config.di_Pos_Window))
                   AND "gtyp_VGR".horizontal_Axis.x_Position_Reached THEN
                   "gtyp_VGR".horizontal_Axis.x_Start_Positioning := FALSE;
                   #li_StepCase := 440;
               END_IF;

           440: // Container Available start pick up
               IF "gtyp_HBW".x_HBW_Container_Available THEN
                   #li_StepCase := 450;
               END_IF;

           450: // Position vertical Collect HBW
               "gtyp_VGR".vertical_Axis.di_Target_Position := "gtyp_VGR".di_Pos_HBW_Collect_vertical;
               "gtyp_VGR".vertical_Axis.x_Start_Positioning := TRUE;
               "gtyp_VGR".vertical_Axis.i_PWM := 500;

               IF ("gtyp_VGR".vertical_Axis.di_Actual_Position <= ("gtyp_VGR".di_Pos_HBW_Collect_vertical + "gtyp_VGR".vertical_Axis.Config.di_Pos_Window))
                   AND ("gtyp_VGR".vertical_Axis.di_Actual_Position >= ("gtyp_VGR".di_Pos_HBW_Collect_vertical - "gtyp_VGR".vertical_Axis.Config.di_Pos_Window))
                   AND "gtyp_VGR".vertical_Axis.x_Position_Reached THEN
                   "gtyp_VGR".vertical_Axis.x_Start_Positioning := FALSE;
                   "gtyp_VGR".vertical_Axis.i_PWM := 800;
                   #li_StepCase := 460;
               END_IF;

           460: // turn on compressor
               "QX_VGR_Compressor_Q7" := TRUE;
               "gtyp_VGR".x_MPO_Req_Discard := TRUE;
               #li_StepCase := 470;

           470: // turn on vacuum
               "QX_VGR_ValveVacuum_Q8" := TRUE;

               #lx_Start_TON_Wait := TRUE;
               #lt_TON_Wait := T#500ms;

               IF #lfb_TON_Wait.Q THEN
                   #lx_Start_TON_Wait := FALSE;
                   #li_StepCase := 480;
               END_IF;

           480: // homing vertical axis

               "gtyp_VGR".vertical_Axis.x_Reference := TRUE;

               IF NOT "gtyp_VGR".vertical_Axis.x_Referenced THEN
                   "gtyp_VGR".x_HBW_PickedUp := TRUE;
                   #li_StepCase := 485;
               END_IF;

           485: // homed vertical axis
               IF "gtyp_VGR".vertical_Axis.x_Referenced THEN
                   "gtyp_VGR".vertical_Axis.x_Reference := FALSE;
                   #li_StepCase := 490;
               END_IF;

           490: // homing horizontal axis

               "gtyp_VGR".horizontal_Axis.x_Reference := TRUE;

               IF NOT "gtyp_VGR".horizontal_Axis.x_Referenced THEN
                   #li_StepCase := 495;
               END_IF;

           495: // homed horizontal axis
               IF "gtyp_VGR".horizontal_Axis.x_Referenced THEN
                   "gtyp_VGR".horizontal_Axis.x_Reference := FALSE;
                   #li_StepCase := 500;
               END_IF;

           500: // wait sequence
               #lx_Start_TON_Wait := TRUE;
               #lt_TON_Wait := T#500ms;

               IF #lfb_TON_Wait.Q THEN
                   #lx_State_activ := TRUE;
                   #ls_Target := 'mpo';
                   "gtyp_VGR".x_HBW_PickedUp := FALSE;
                   #lx_Start_TON_Wait := FALSE;
                   #li_StepCase := 510;
               END_IF;

           510: // Position rotate MPO

               "gtyp_VGR".rotate_Axis.di_Target_Position := "gtyp_VGR".di_Pos_MPO_rotate;
               "gtyp_VGR".rotate_Axis.x_Start_Positioning := TRUE;

               IF ("gtyp_VGR".rotate_Axis.di_Actual_Position <= ("gtyp_VGR".di_Pos_MPO_rotate + "gtyp_VGR".rotate_Axis.Config.di_Pos_Window))
                   AND ("gtyp_VGR".rotate_Axis.di_Actual_Position >= ("gtyp_VGR".di_Pos_MPO_rotate - "gtyp_VGR".rotate_Axis.Config.di_Pos_Window))
                   AND "gtyp_VGR".rotate_Axis.x_Position_Reached THEN
                   "gtyp_VGR".rotate_Axis.x_Start_Positioning := FALSE;
                   #li_StepCase := 515;
               END_IF;

           515: // Position horizontal/pre vertical MPO

               "gtyp_VGR".horizontal_Axis.di_Target_Position := "gtyp_VGR".di_Pos_MPO_horizontal;
               "gtyp_VGR".horizontal_Axis.x_Start_Positioning := TRUE;
               "gtyp_VGR".vertical_Axis.di_Target_Position := "gtyp_VGR".di_Pos_MPO_vertical - "gtyp_VGR".di_Offset_Pos_MPO_vertical;
               "gtyp_VGR".vertical_Axis.x_Start_Positioning := TRUE;
               "gtyp_VGR".vertical_Axis.i_PWM := 500;

               IF ("gtyp_VGR".horizontal_Axis.di_Actual_Position <= ("gtyp_VGR".di_Pos_MPO_horizontal + "gtyp_VGR".horizontal_Axis.Config.di_Pos_Window))
                   AND ("gtyp_VGR".horizontal_Axis.di_Actual_Position >= ("gtyp_VGR".di_Pos_MPO_horizontal - "gtyp_VGR".horizontal_Axis.Config.di_Pos_Window))
                   AND "gtyp_VGR".horizontal_Axis.x_Position_Reached THEN
                   "gtyp_VGR".horizontal_Axis.x_Start_Positioning := FALSE;
               END_IF;

               IF ("gtyp_VGR".vertical_Axis.di_Actual_Position <= ("gtyp_VGR".di_Pos_MPO_vertical - "gtyp_VGR".di_Offset_Pos_MPO_vertical + "gtyp_VGR".vertical_Axis.Config.di_Pos_Window))
                   AND ("gtyp_VGR".vertical_Axis.di_Actual_Position >= ("gtyp_VGR".di_Pos_MPO_vertical - "gtyp_VGR".di_Offset_Pos_MPO_vertical - "gtyp_VGR".vertical_Axis.Config.di_Pos_Window))
                   AND "gtyp_VGR".vertical_Axis.x_Position_Reached THEN
                   "gtyp_VGR".vertical_Axis.x_Start_Positioning := FALSE;
               END_IF;

               IF ("gtyp_VGR".horizontal_Axis.di_Actual_Position <= ("gtyp_VGR".di_Pos_MPO_horizontal + "gtyp_VGR".horizontal_Axis.Config.di_Pos_Window))
                   AND ("gtyp_VGR".horizontal_Axis.di_Actual_Position >= ("gtyp_VGR".di_Pos_MPO_horizontal - "gtyp_VGR".horizontal_Axis.Config.di_Pos_Window))
                   AND "gtyp_VGR".horizontal_Axis.x_Position_Reached
                   AND ("gtyp_VGR".vertical_Axis.di_Actual_Position <= ("gtyp_VGR".di_Pos_MPO_vertical - "gtyp_VGR".di_Offset_Pos_MPO_vertical + "gtyp_VGR".vertical_Axis.Config.di_Pos_Window))
                   AND ("gtyp_VGR".vertical_Axis.di_Actual_Position >= ("gtyp_VGR".di_Pos_MPO_vertical - "gtyp_VGR".di_Offset_Pos_MPO_vertical - "gtyp_VGR".vertical_Axis.Config.di_Pos_Window))
                   AND "gtyp_VGR".vertical_Axis.x_Position_Reached THEN
                   "gtyp_VGR".horizontal_Axis.x_Start_Positioning := FALSE;
                   "gtyp_VGR".vertical_Axis.x_Start_Positioning := FALSE;
                   "gtyp_VGR".vertical_Axis.i_PWM := 800;
                   #li_StepCase := 520;
               END_IF;

           520: // MPO ready to discard - Position vertical MPO

               IF "gtyp_MPO".x_Discard_Ready THEN
                   "gtyp_VGR".vertical_Axis.di_Target_Position := "gtyp_VGR".di_Pos_MPO_vertical;
                   "gtyp_VGR".vertical_Axis.x_Start_Positioning := TRUE;
                   "gtyp_VGR".vertical_Axis.i_PWM := 500;

                   IF ("gtyp_VGR".vertical_Axis.di_Actual_Position <= ("gtyp_VGR".di_Pos_MPO_vertical + "gtyp_VGR".vertical_Axis.Config.di_Pos_Window))
                       AND ("gtyp_VGR".vertical_Axis.di_Actual_Position >= ("gtyp_VGR".di_Pos_MPO_vertical - "gtyp_VGR".vertical_Axis.Config.di_Pos_Window))
                       AND "gtyp_VGR".vertical_Axis.x_Position_Reached THEN
                       "gtyp_VGR".vertical_Axis.x_Start_Positioning := FALSE;
                       "gtyp_VGR".vertical_Axis.i_PWM := 800;
                       #li_StepCase := 530;
                       "gtyp_VGR".x_MPO_Req_Discard := FALSE;
                   END_IF;
               END_IF;

           530: // turn off vacuum
               "QX_VGR_ValveVacuum_Q8" := FALSE;
               #li_StepCase := 540;

           540: // turn off compressor
               "QX_VGR_Compressor_Q7" := FALSE;
               "gtyp_VGR".x_MPO_Discards := TRUE;
               // Order State
               "gtyp_VGR".x_Ready_For_Outsource := FALSE;
               "gtyp_VGR".x_State_Process := TRUE;
               "gtyp_Interface_Dashboard".Subscribe.State_Order.ldt_ts := DT_TO_LDT(#ldt_MQTT);
               "gtyp_Interface_Dashboard".Subscribe.State_Order.s_state := 'IN_PROCESS';
               "gtyp_Interface_Dashboard".Subscribe.State_Order.s_type := "gtyp_VGR".Workpiece.s_type;
               #li_StepCase := 550;

           550: // Workpiece discard accepted - Position pre vertical MPO

               IF "gtyp_MPO".x_MPO_Discards_Accepted THEN
                   "gtyp_VGR".vertical_Axis.di_Target_Position := "gtyp_VGR".di_Pos_MPO_vertical - "gtyp_VGR".di_Offset_Pos_MPO_vertical;
                   "gtyp_VGR".vertical_Axis.x_Start_Positioning := TRUE;
                   "gtyp_VGR".vertical_Axis.i_PWM := 500;

                   IF ("gtyp_VGR".vertical_Axis.di_Actual_Position <= ("gtyp_VGR".di_Pos_MPO_vertical - "gtyp_VGR".di_Offset_Pos_MPO_vertical + "gtyp_VGR".vertical_Axis.Config.di_Pos_Window))
                       AND ("gtyp_VGR".vertical_Axis.di_Actual_Position >= ("gtyp_VGR".di_Pos_MPO_vertical - "gtyp_VGR".di_Offset_Pos_MPO_vertical - "gtyp_VGR".vertical_Axis.Config.di_Pos_Window))
                       AND "gtyp_VGR".vertical_Axis.x_Position_Reached THEN
                       "gtyp_VGR".vertical_Axis.x_Start_Positioning := FALSE;
                       "gtyp_VGR".x_MPO_Discards := FALSE;
                       "gtyp_VGR".vertical_Axis.i_PWM := 800;
                       #li_StepCase := 560;
                   END_IF;
               END_IF;

           560: // homing horizontal axis
               "gtyp_VGR".horizontal_Axis.x_Reference := TRUE;

               IF NOT "gtyp_VGR".horizontal_Axis.x_Referenced THEN
                   #li_StepCase := 570;
               END_IF;

           570: // homed horizontal axis
               IF "gtyp_VGR".horizontal_Axis.x_Referenced THEN
                   "gtyp_VGR".horizontal_Axis.x_Reference := FALSE;
                   "gtyp_VGR".x_MPO_Discards := FALSE;
                   #li_StepCase := 580;
               END_IF;

           580: // wait sequence
               #lx_Start_TON_Wait := TRUE;
               #lt_TON_Wait := T#500ms;

               IF #lfb_TON_Wait.Q THEN
                   "gtyp_VGR".Workpiece.s_id := '0';
                   "gtyp_VGR".Workpiece.s_state := '';
                   "gtyp_VGR".Workpiece.s_type := '';
                   FOR #li_Counter := 1 TO 8 DO
                       "gtyp_VGR".History[#li_Counter].i_code := 0;
                       "gtyp_VGR".History[#li_Counter].ldt_ts := DT#1990-01-01-00:00:00;
                   END_FOR;
                   #lx_Start_TON_Wait := FALSE;
                   #li_StepCase := 0;
               END_IF;

               (*******************************************************************************************)
               (**************************      Procedure - store raw parts      **************************)
               (*******************************************************************************************)

           600:// approach pick-up position dsi with vertical, horizontal, rotate axis
               "gtyp_VGR".horizontal_Axis.di_Target_Position := "gtyp_VGR".di_Pos_DSI_horizontal;
               "gtyp_VGR".horizontal_Axis.x_Start_Positioning := TRUE;
               "gtyp_VGR".vertical_Axis.di_Target_Position := "gtyp_VGR".di_Pos_DSI_Collect_vertical;
               "gtyp_VGR".vertical_Axis.x_Start_Positioning := TRUE;
               "gtyp_VGR".vertical_Axis.i_PWM := 500;
               "gtyp_VGR".rotate_Axis.di_Target_Position := "gtyp_VGR".di_Pos_DSI_rotate;
               "gtyp_VGR".rotate_Axis.x_Start_Positioning := TRUE;

               IF ("gtyp_VGR".horizontal_Axis.di_Actual_Position <= ("gtyp_VGR".di_Pos_DSI_horizontal + "gtyp_VGR".horizontal_Axis.Config.di_Pos_Window))
                   AND ("gtyp_VGR".horizontal_Axis.di_Actual_Position >= ("gtyp_VGR".di_Pos_DSI_horizontal - "gtyp_VGR".horizontal_Axis.Config.di_Pos_Window))
                   AND "gtyp_VGR".horizontal_Axis.x_Position_Reached THEN
                   "gtyp_VGR".horizontal_Axis.x_Start_Positioning := FALSE;
               END_IF;

               IF ("gtyp_VGR".vertical_Axis.di_Actual_Position <= ("gtyp_VGR".di_Pos_DSI_Collect_vertical + "gtyp_VGR".vertical_Axis.Config.di_Pos_Window))
                   AND ("gtyp_VGR".vertical_Axis.di_Actual_Position >= ("gtyp_VGR".di_Pos_DSI_Collect_vertical - "gtyp_VGR".vertical_Axis.Config.di_Pos_Window))
                   AND "gtyp_VGR".vertical_Axis.x_Position_Reached THEN
                   "gtyp_VGR".vertical_Axis.x_Start_Positioning := FALSE;
               END_IF;

               IF ("gtyp_VGR".rotate_Axis.di_Actual_Position <= ("gtyp_VGR".di_Pos_DSI_rotate + "gtyp_VGR".rotate_Axis.Config.di_Pos_Window))
                   AND ("gtyp_VGR".rotate_Axis.di_Actual_Position >= ("gtyp_VGR".di_Pos_DSI_rotate - "gtyp_VGR".rotate_Axis.Config.di_Pos_Window))
                   AND "gtyp_VGR".rotate_Axis.x_Position_Reached THEN
                   "gtyp_VGR".rotate_Axis.x_Start_Positioning := FALSE;
               END_IF;

               IF ("gtyp_VGR".horizontal_Axis.di_Actual_Position <= ("gtyp_VGR".di_Pos_DSI_horizontal + "gtyp_VGR".horizontal_Axis.Config.di_Pos_Window))
                   AND ("gtyp_VGR".horizontal_Axis.di_Actual_Position >= ("gtyp_VGR".di_Pos_DSI_horizontal - "gtyp_VGR".horizontal_Axis.Config.di_Pos_Window))
                   AND "gtyp_VGR".horizontal_Axis.x_Position_Reached
                   AND ("gtyp_VGR".vertical_Axis.di_Actual_Position <= ("gtyp_VGR".di_Pos_DSI_Collect_vertical + "gtyp_VGR".vertical_Axis.Config.di_Pos_Window))
                   AND ("gtyp_VGR".vertical_Axis.di_Actual_Position >= ("gtyp_VGR".di_Pos_DSI_Collect_vertical - "gtyp_VGR".vertical_Axis.Config.di_Pos_Window))
                   AND "gtyp_VGR".vertical_Axis.x_Position_Reached
                   AND ("gtyp_VGR".rotate_Axis.di_Actual_Position <= ("gtyp_VGR".di_Pos_DSI_rotate + "gtyp_VGR".rotate_Axis.Config.di_Pos_Window))
                   AND ("gtyp_VGR".rotate_Axis.di_Actual_Position >= ("gtyp_VGR".di_Pos_DSI_rotate - "gtyp_VGR".rotate_Axis.Config.di_Pos_Window))
                   AND "gtyp_VGR".rotate_Axis.x_Position_Reached THEN
                   "gtyp_VGR".horizontal_Axis.x_Start_Positioning := FALSE;
                   "gtyp_VGR".vertical_Axis.x_Start_Positioning := FALSE;
                   "gtyp_VGR".rotate_Axis.x_Start_Positioning := FALSE;
                   "gtyp_VGR".vertical_Axis.i_PWM := 800;
                   #li_StepCase := 610;
               END_IF;

           610:// set status 100 raw goods delivered
               #li_Return_LDT := RD_SYS_T(#ldt_MQTT);
               "gtyp_VGR".Workpiece.s_state := 'RAW';
               "gtyp_VGR".History[1].ldt_ts := DT_TO_LDT(#ldt_MQTT);
               "gtyp_VGR".History[1].i_code := 100;
               #li_StepCase := 620;

           620:// wait sequence
               #lx_Start_TON_Wait := TRUE;
               #lt_TON_Wait := T#500ms;

               IF #lfb_TON_Wait.Q THEN
                   #lx_Start_TON_Wait := FALSE;
                   #li_StepCase := 630;
               END_IF;

           630:// turn on compressor and wait
               "QX_VGR_Compressor_Q7" := TRUE;

               #lx_Start_TON_Wait := TRUE;
               #lt_TON_Wait := T#500ms;

               IF #lfb_TON_Wait.Q THEN
                   #lx_Start_TON_Wait := FALSE;
                   #li_StepCase := 640;
               END_IF;

           640:// turn on vacuum 
               "QX_VGR_ValveVacuum_Q8" := true;

               #li_StepCase := 650;

           650:// Position vertical NFC
               #lx_State_activ := TRUE;
               #ls_Target := 'hbw';

               "gtyp_VGR".vertical_Axis.di_Target_Position := "gtyp_VGR".di_Pos_NFC_vertical - "gtyp_VGR".di_Offset_Pos_DSI_NFC_vertical;
               "gtyp_VGR".vertical_Axis.x_Start_Positioning := TRUE;
               "gtyp_VGR".vertical_Axis.i_PWM := 800;

               IF ("gtyp_VGR".vertical_Axis.di_Actual_Position <= ("gtyp_VGR".di_Pos_NFC_vertical - "gtyp_VGR".di_Offset_Pos_DSI_NFC_vertical + "gtyp_VGR".vertical_Axis.Config.di_Pos_Window))
                   AND ("gtyp_VGR".vertical_Axis.di_Actual_Position >= ("gtyp_VGR".di_Pos_NFC_vertical - "gtyp_VGR".di_Offset_Pos_DSI_NFC_vertical - "gtyp_VGR".vertical_Axis.Config.di_Pos_Window))
                   AND "gtyp_VGR".vertical_Axis.x_Position_Reached THEN
                   "gtyp_VGR".vertical_Axis.x_Start_Positioning := FALSE;
                   #li_StepCase := 660;
               END_IF;

           660: // wait sequence
               #lx_Start_TON_Wait := TRUE;
               #lt_TON_Wait := T#500ms;

               IF #lfb_TON_Wait.Q THEN
                   #lx_Start_TON_Wait := FALSE;
                   #li_StepCase := 670;
               END_IF;

           670: // Position horizontal/rotate NFC

               "gtyp_VGR".horizontal_Axis.di_Target_Position := "gtyp_VGR".di_Pos_NFC_horizontal;
               "gtyp_VGR".horizontal_Axis.x_Start_Positioning := TRUE;
               "gtyp_VGR".rotate_Axis.di_Target_Position := "gtyp_VGR".di_Pos_NFC_rotate;
               "gtyp_VGR".rotate_Axis.x_Start_Positioning := TRUE;

               IF ("gtyp_VGR".horizontal_Axis.di_Actual_Position <= ("gtyp_VGR".di_Pos_NFC_horizontal + "gtyp_VGR".horizontal_Axis.Config.di_Pos_Window))
                   AND ("gtyp_VGR".horizontal_Axis.di_Actual_Position >= ("gtyp_VGR".di_Pos_NFC_horizontal - "gtyp_VGR".horizontal_Axis.Config.di_Pos_Window))
                   AND "gtyp_VGR".horizontal_Axis.x_Position_Reached THEN
                   "gtyp_VGR".horizontal_Axis.x_Start_Positioning := FALSE;
               END_IF;

               IF ("gtyp_VGR".rotate_Axis.di_Actual_Position <= ("gtyp_VGR".di_Pos_NFC_rotate + "gtyp_VGR".rotate_Axis.Config.di_Pos_Window))
                   AND ("gtyp_VGR".rotate_Axis.di_Actual_Position >= ("gtyp_VGR".di_Pos_NFC_rotate - "gtyp_VGR".rotate_Axis.Config.di_Pos_Window))
                   AND "gtyp_VGR".rotate_Axis.x_Position_Reached THEN
                   "gtyp_VGR".rotate_Axis.x_Start_Positioning := FALSE;
               END_IF;

               IF ("gtyp_VGR".horizontal_Axis.di_Actual_Position <= ("gtyp_VGR".di_Pos_NFC_horizontal + "gtyp_VGR".horizontal_Axis.Config.di_Pos_Window))
                   AND ("gtyp_VGR".horizontal_Axis.di_Actual_Position >= ("gtyp_VGR".di_Pos_NFC_horizontal - "gtyp_VGR".horizontal_Axis.Config.di_Pos_Window))
                   AND "gtyp_VGR".horizontal_Axis.x_Position_Reached
                   AND ("gtyp_VGR".rotate_Axis.di_Actual_Position <= ("gtyp_VGR".di_Pos_NFC_rotate + "gtyp_VGR".rotate_Axis.Config.di_Pos_Window))
                   AND ("gtyp_VGR".rotate_Axis.di_Actual_Position >= ("gtyp_VGR".di_Pos_NFC_rotate - "gtyp_VGR".rotate_Axis.Config.di_Pos_Window))
                   AND "gtyp_VGR".rotate_Axis.x_Position_Reached THEN
                   "gtyp_VGR".horizontal_Axis.x_Start_Positioning := FALSE;
                   "gtyp_VGR".rotate_Axis.x_Start_Positioning := FALSE;
                   #li_StepCase := 680;
               END_IF;

           680: // wait sequence
               #lx_Start_TON_Wait := TRUE;
               #lt_TON_Wait := T#500ms;

               IF #lfb_TON_Wait.Q THEN
                   #lx_Start_TON_Wait := FALSE;
                   #li_StepCase := 690;
               END_IF;

           690: // Position vertical NFC

               "gtyp_VGR".vertical_Axis.di_Target_Position := "gtyp_VGR".di_Pos_NFC_vertical;
               "gtyp_VGR".vertical_Axis.x_Start_Positioning := TRUE;
               "gtyp_VGR".vertical_Axis.i_PWM := 500;

               IF ("gtyp_VGR".vertical_Axis.di_Actual_Position <= ("gtyp_VGR".di_Pos_NFC_vertical + "gtyp_VGR".vertical_Axis.Config.di_Pos_Window))
                   AND ("gtyp_VGR".vertical_Axis.di_Actual_Position >= ("gtyp_VGR".di_Pos_NFC_vertical - "gtyp_VGR".vertical_Axis.Config.di_Pos_Window))
                   AND "gtyp_VGR".vertical_Axis.x_Position_Reached THEN
                   "gtyp_VGR".vertical_Axis.x_Start_Positioning := FALSE;
                   "gtyp_VGR".vertical_Axis.i_PWM := 800;
                   #li_StepCase := 700;
               END_IF;

           700: // Start delete/write/read NFC 
               "gtyp_VGR".x_NFC_Start_First := TRUE;

               IF "gtyp_VGR".x_NFC_Completed THEN
                   "gtyp_VGR".x_NFC_Start_First := FALSE;
                   #li_StepCase := 710;
               END_IF;

           710: // Position vertical pre NFC

               "gtyp_VGR".vertical_Axis.di_Target_Position := "gtyp_VGR".di_Pos_NFC_vertical - "gtyp_VGR".di_Offset_Pos_DSI_NFC_vertical;
               "gtyp_VGR".vertical_Axis.x_Start_Positioning := TRUE;
               "gtyp_VGR".vertical_Axis.i_PWM := 800;

               IF ("gtyp_VGR".vertical_Axis.di_Actual_Position <= ("gtyp_VGR".di_Pos_NFC_vertical - "gtyp_VGR".di_Offset_Pos_DSI_NFC_vertical + "gtyp_VGR".vertical_Axis.Config.di_Pos_Window))
                   AND ("gtyp_VGR".vertical_Axis.di_Actual_Position >= ("gtyp_VGR".di_Pos_NFC_vertical - "gtyp_VGR".di_Offset_Pos_DSI_NFC_vertical - "gtyp_VGR".vertical_Axis.Config.di_Pos_Window))
                   AND "gtyp_VGR".vertical_Axis.x_Position_Reached THEN
                   "gtyp_VGR".vertical_Axis.x_Start_Positioning := FALSE;
                   #li_StepCase := 720;
               END_IF;

           720: // Position horizontal/rotate Color

               "gtyp_VGR".horizontal_Axis.di_Target_Position := "gtyp_VGR".di_Pos_Color_horizontal;
               "gtyp_VGR".horizontal_Axis.x_Start_Positioning := TRUE;
               "gtyp_VGR".rotate_Axis.di_Target_Position := "gtyp_VGR".di_Pos_Color_rotate;
               "gtyp_VGR".rotate_Axis.x_Start_Positioning := TRUE;

               IF ("gtyp_VGR".horizontal_Axis.di_Actual_Position <= ("gtyp_VGR".di_Pos_Color_horizontal + "gtyp_VGR".horizontal_Axis.Config.di_Pos_Window))
                   AND ("gtyp_VGR".horizontal_Axis.di_Actual_Position >= ("gtyp_VGR".di_Pos_Color_horizontal - "gtyp_VGR".horizontal_Axis.Config.di_Pos_Window))
                   AND "gtyp_VGR".horizontal_Axis.x_Position_Reached THEN
                   "gtyp_VGR".horizontal_Axis.x_Start_Positioning := FALSE;
               END_IF;

               IF ("gtyp_VGR".rotate_Axis.di_Actual_Position <= ("gtyp_VGR".di_Pos_Color_rotate + "gtyp_VGR".rotate_Axis.Config.di_Pos_Window))
                   AND ("gtyp_VGR".rotate_Axis.di_Actual_Position >= ("gtyp_VGR".di_Pos_Color_rotate - "gtyp_VGR".rotate_Axis.Config.di_Pos_Window))
                   AND "gtyp_VGR".rotate_Axis.x_Position_Reached THEN
                   "gtyp_VGR".rotate_Axis.x_Start_Positioning := FALSE;
               END_IF;

               IF ("gtyp_VGR".horizontal_Axis.di_Actual_Position <= ("gtyp_VGR".di_Pos_Color_horizontal + "gtyp_VGR".horizontal_Axis.Config.di_Pos_Window))
                   AND ("gtyp_VGR".horizontal_Axis.di_Actual_Position >= ("gtyp_VGR".di_Pos_Color_horizontal - "gtyp_VGR".horizontal_Axis.Config.di_Pos_Window))
                   AND "gtyp_VGR".horizontal_Axis.x_Position_Reached
                   AND ("gtyp_VGR".rotate_Axis.di_Actual_Position <= ("gtyp_VGR".di_Pos_Color_rotate + "gtyp_VGR".rotate_Axis.Config.di_Pos_Window))
                   AND ("gtyp_VGR".rotate_Axis.di_Actual_Position >= ("gtyp_VGR".di_Pos_Color_rotate - "gtyp_VGR".rotate_Axis.Config.di_Pos_Window))
                   AND "gtyp_VGR".rotate_Axis.x_Position_Reached THEN
                   "gtyp_VGR".horizontal_Axis.x_Start_Positioning := FALSE;
                   "gtyp_VGR".rotate_Axis.x_Start_Positioning := FALSE;
                   #li_StepCase := 730;
               END_IF;

           730: // wait sequence
               #lx_Start_TON_Wait := TRUE;
               #lt_TON_Wait := T#500ms;

               IF #lfb_TON_Wait.Q THEN
                   #lx_Start_TON_Wait := FALSE;
                   #li_StepCase := 740;
               END_IF;

           740: // Position vertical Color
               "gtyp_VGR".vertical_Axis.di_Target_Position := "gtyp_VGR".di_Pos_Color_vertical;
               "gtyp_VGR".vertical_Axis.x_Start_Positioning := TRUE;
               "gtyp_VGR".vertical_Axis.i_PWM := 500;

